LIN {X 0,Y 525.435,Z 278.246,A -85,B 0,C 180,E1 -4754.99,E2 -4754.99} C_VEL
LIN {X 0,Y 525.931,Z 282.457,A -85,B 0,C 180,E1 -4755.064,E2 -4755.064} C_VEL
LIN {X 0,Y 525.504,Z 378.759,A -85,B 0,C 180,E1 -4756.414,E2 -4756.414} C_VEL
LIN {X 0,Y 525.272,Z 391.955,A -85,B 0,C 180,E1 -4756.753,E2 -4756.753} C_VEL
LIN {X 0,Y 525.033,Z 404.647,A -85,B 0,C 180,E1 -4757.239,E2 -4757.239} C_VEL
LIN {X 0,Y 524.762,Z 415.969,A -85,B 0,C 180,E1 -4757.824,E2 -4757.824} C_VEL
LIN {X 0,Y 524.543,Z 427.589,A -85,B 0,C 180,E1 -4758.601,E2 -4758.601} C_VEL
LIN {X 0,Y 524.212,Z 438.073,A -85,B 0,C 180,E1 -4759.474,E2 -4759.474} C_VEL
LIN {X 0,Y 524.018,Z 446.642,A -85,B 0,C 180,E1 -4760.348,E2 -4760.348} C_VEL
LIN {X 0,Y 523.819,Z 454.543,A -85,B 0,C 180,E1 -4761.317,E2 -4761.317} C_VEL
LIN {X 0,Y 523.627,Z 462.256,A -85,B 0,C 180,E1 -4762.479,E2 -4762.479} C_VEL
LIN {X 0,Y 523.496,Z 469.355,A -85,B 0,C 180,E1 -4763.833,E2 -4763.833} C_VEL
LIN {X 0,Y 523.385,Z 474.077,A -85,B 0,C 180,E1 -4764.992,E2 -4764.992} C_VEL
LIN {X 0,Y 523.446,Z 477.686,A -85,B 0,C 180,E1 -4766.149,E2 -4766.149} C_VEL
LIN {X 0,Y 523.37,Z 479.546,A -85,B 0,C 180,E1 -4766.92,E2 -4766.92} C_VEL
LIN {X 0,Y 523.336,Z 480.94,A -85,B 0,C 180,E1 -4767.69,E2 -4767.69} C_VEL
LIN {X 0,Y 523.251,Z 482.541,A -85,B 0,C 180,E1 -4769.229,E2 -4769.229} C_VEL
LIN {X 0,Y 523.248,Z 482.758,A -85,B 0,C 180,E1 -4769.999,E2 -4769.999} C_VEL
LIN {X 0,Y 523.275,Z 481.936,A -85,B 0,C 180,E1 -4771.538,E2 -4771.538} C_VEL
LIN {X 0,Y 523.336,Z 480.943,A -85,B 0,C 180,E1 -4772.308,E2 -4772.308} C_VEL
LIN {X 0,Y 523.369,Z 479.548,A -85,B 0,C 180,E1 -4773.078,E2 -4773.078} C_VEL
LIN {X 0,Y 523.425,Z 476.616,A -85,B 0,C 180,E1 -4774.234,E2 -4774.234} C_VEL
LIN {X 0,Y 523.461,Z 472.643,A -85,B 0,C 180,E1 -4775.391,E2 -4775.391} C_VEL
LIN {X 0,Y 523.504,Z 466.574,A -85,B 0,C 180,E1 -4776.736,E2 -4776.736} C_VEL
LIN {X 0,Y 523.675,Z 459.848,A -85,B 0,C 180,E1 -4777.905,E2 -4777.905} C_VEL
LIN {X 0,Y 523.855,Z 451.549,A -85,B 0,C 180,E1 -4779.068,E2 -4779.068} C_VEL
LIN {X 0,Y 524.068,Z 443.032,A -85,B 0,C 180,E1 -4780.039,E2 -4780.039} C_VEL
LIN {X 0,Y 524.349,Z 432.504,A -85,B 0,C 180,E1 -4781.009,E2 -4781.009} C_VEL
LIN {X 0,Y 524.658,Z 422.256,A -85,B 0,C 180,E1 -4781.774,E2 -4781.774} C_VEL
LIN {X 0,Y 524.908,Z 410.629,A -85,B 0,C 180,E1 -4782.467,E2 -4782.467} C_VEL
LIN {X 0,Y 525.182,Z 398.8,A -85,B 0,C 180,E1 -4783,E2 -4783} C_VEL
LIN {X 0,Y 525.389,Z 386.064,A -85,B 0,C 180,E1 -4783.413,E2 -4783.413} C_VEL
LIN {X 0,Y 525.543,Z 372.951,A -85,B 0,C 180,E1 -4783.68,E2 -4783.68} C_VEL
LIN {X 0,Y 525.872,Z 280.781,A -85,B 0,C 180,E1 -4784.959,E2 -4784.959} C_VEL
LIN {X 0,Y 524.29,Z 270.778,A -85,B 0,C 180,E1 -4785.168,E2 -4785.168} C_VEL
LIN {X 0,Y 524.631,Z 252.415,A -85,B 0,C 180,E1 -4788.125,E2 -4788.125} C_VEL
LIN {X 0,Y 525.085,Z 232.615,A -85,B 0,C 180,E1 -4791.389,E2 -4791.389} C_VEL
LIN {X 0,Y 524.921,Z 226.943,A -85,B 0,C 180,E1 -4792.346,E2 -4792.346} C_VEL
LIN {X 0,Y 524.015,Z 222.139,A -85,B 0,C 180,E1 -4793.2,E2 -4793.2} C_VEL
LIN {X 0,Y 523.924,Z 221.726,A -85,B 0,C 180,E1 -4793.414,E2 -4793.414} C_VEL
LIN {X 0,Y 523.946,Z 221.719,A -85,B 0,C 180,E1 -4796.271,E2 -4796.271} C_VEL
LIN {X 0,Y 523.933,Z 221.718,A -85,B 0,C 180,E1 -4798.873,E2 -4798.873} C_VEL
LIN {X 0,Y 523.923,Z 221.722,A -85,B 0,C 180,E1 -4801.542,E2 -4801.542} C_VEL
LIN {X 0,Y 523.934,Z 221.721,A -85,B 0,C 180,E1 -4804.288,E2 -4804.288} C_VEL
LIN {X 0,Y 523.906,Z 221.721,A -85,B 0,C 180,E1 -4807.13,E2 -4807.13} C_VEL
LIN {X 0,Y 523.915,Z 221.727,A -85,B 0,C 180,E1 -4810.124,E2 -4810.124} C_VEL
LIN {X 0,Y 523.887,Z 221.721,A -85,B 0,C 180,E1 -4813.168,E2 -4813.168} C_VEL
LIN {X 0,Y 523.919,Z 221.721,A -85,B 0,C 180,E1 -4815.767,E2 -4815.767} C_VEL
LIN {X 0,Y 523.896,Z 221.723,A -85,B 0,C 180,E1 -4818.9,E2 -4818.9} C_VEL
LIN {X 0,Y 523.899,Z 221.723,A -85,B 0,C 180,E1 -4821.894,E2 -4821.894} C_VEL
LIN {X 0,Y 523.914,Z 221.722,A -85,B 0,C 180,E1 -4824.909,E2 -4824.909} C_VEL
LIN {X 0,Y 523.929,Z 221.716,A -85,B 0,C 180,E1 -4827.677,E2 -4827.677} C_VEL
LIN {X 0,Y 523.932,Z 221.724,A -85,B 0,C 180,E1 -4830.677,E2 -4830.677} C_VEL
LIN {X 0,Y 523.893,Z 221.719,A -85,B 0,C 180,E1 -4833.721,E2 -4833.721} C_VEL
LIN {X 0,Y 523.889,Z 221.725,A -85,B 0,C 180,E1 -4836.265,E2 -4836.265} C_VEL
LIN {X 0,Y 523.908,Z 221.729,A -85,B 0,C 180,E1 -4838.761,E2 -4838.761} C_VEL
LIN {X 0,Y 523.907,Z 221.723,A -85,B 0,C 180,E1 -4841.215,E2 -4841.215} C_VEL
LIN {X 0,Y 523.867,Z 221.724,A -85,B 0,C 180,E1 -4843.633,E2 -4843.633} C_VEL
LIN {X 0,Y 523.95,Z 221.719,A -85,B 0,C 180,E1 -4845.231,E2 -4845.231} C_VEL
LIN {X 0,Y 523.983,Z 221.71,A -85,B 0,C 180,E1 -4848.389,E2 -4848.389} C_VEL
LIN {X 0,Y 523.936,Z 221.719,A -85,B 0,C 180,E1 -4851.51,E2 -4851.51} C_VEL
LIN {X 0,Y 523.997,Z 221.708,A -85,B 0,C 180,E1 -4853.836,E2 -4853.836} C_VEL
LIN {X 0,Y 524.014,Z 221.712,A -85,B 0,C 180,E1 -4856.92,E2 -4856.92} C_VEL
LIN {X 0,Y 524.088,Z 221.697,A -85,B 0,C 180,E1 -4859.995,E2 -4859.995} C_VEL
LIN {X 0,Y 524.048,Z 221.707,A -85,B 0,C 180,E1 -4863.07,E2 -4863.07} C_VEL
LIN {X 0,Y 524.011,Z 221.708,A -85,B 0,C 180,E1 -4866.154,E2 -4866.154} C_VEL
LIN {X 0,Y 523.979,Z 221.711,A -85,B 0,C 180,E1 -4868.479,E2 -4868.479} C_VEL
LIN {X 0,Y 523.997,Z 221.716,A -85,B 0,C 180,E1 -4871.746,E2 -4871.746} C_VEL
LIN {X 0,Y 523.963,Z 221.715,A -85,B 0,C 180,E1 -4875.048,E2 -4875.048} C_VEL
LIN {X 0,Y 523.931,Z 221.724,A -85,B 0,C 180,E1 -4877.964,E2 -4877.964} C_VEL
LIN {X 0,Y 523.938,Z 221.718,A -85,B 0,C 180,E1 -4880.405,E2 -4880.405} C_VEL
LIN {X 0,Y 523.927,Z 221.72,A -85,B 0,C 180,E1 -4882.886,E2 -4882.886} C_VEL
LIN {X 0,Y 524.021,Z 221.823,A -85,B 0,C 180,E1 -4884.93,E2 -4884.93} C_VEL
LIN {X 0,Y 524.568,Z 226.394,A -85,B 0,C 180,E1 -4885.76,E2 -4885.76} C_VEL
LIN {X 0,Y 524.321,Z 244.865,A -85,B 0,C 180,E1 -4888.844,E2 -4888.844} C_VEL
LIN {X 0,Y 524.2,Z 257.025,A -85,B 0,C 180,E1 -4890.872,E2 -4890.872} C_VEL
LIN {X 0,Y 525.251,Z 263.257,A -85,B 0,C 180,E1 -4891.016,E2 -4891.016} C_VEL
LIN {X 0,Y 525.911,Z 268.568,A -85,B 0,C 180,E1 -4891.111,E2 -4891.111} C_VEL
LIN {X 0,Y 525.501,Z 364.681,A -85,B 0,C 180,E1 -4892.465,E2 -4892.465} C_VEL
LIN {X 0,Y 525.441,Z 368.257,A -85,B 0,C 180,E1 -4892.54,E2 -4892.54} C_VEL
LIN {X 0,Y 524.652,Z 374.018,A -85,B 0,C 180,E1 -4892.662,E2 -4892.662} C_VEL
LIN {X 0,Y 521.72,Z 383.263,A -85,B 0,C 180,E1 -4892.894,E2 -4892.894} C_VEL
LIN {X 0,Y 518.781,Z 392.251,A -85,B 0,C 180,E1 -4893.214,E2 -4893.214} C_VEL
LIN {X 0,Y 517.98,Z 397.6,A -85,B 0,C 180,E1 -4893.474,E2 -4893.474} C_VEL
LIN {X 0,Y 517.687,Z 409.287,A -85,B 0,C 180,E1 -4894.194,E2 -4894.194} C_VEL
LIN {X 0,Y 517.367,Z 419.582,A -85,B 0,C 180,E1 -4894.992,E2 -4894.992} C_VEL
LIN {X 0,Y 517.046,Z 430.003,A -85,B 0,C 180,E1 -4895.997,E2 -4895.997} C_VEL
LIN {X 0,Y 516.831,Z 438.296,A -85,B 0,C 180,E1 -4896.984,E2 -4896.984} C_VEL
LIN {X 0,Y 516.612,Z 445.81,A -85,B 0,C 180,E1 -4898.073,E2 -4898.073} C_VEL
LIN {X 0,Y 516.482,Z 451.883,A -85,B 0,C 180,E1 -4899.141,E2 -4899.141} C_VEL
LIN {X 0,Y 516.356,Z 457.376,A -85,B 0,C 180,E1 -4900.344,E2 -4900.344} C_VEL
LIN {X 0,Y 516.321,Z 461.562,A -85,B 0,C 180,E1 -4901.53,E2 -4901.53} C_VEL
LIN {X 0,Y 516.21,Z 465.087,A -85,B 0,C 180,E1 -4902.89,E2 -4902.89} C_VEL
LIN {X 0,Y 516.174,Z 466.943,A -85,B 0,C 180,E1 -4903.968,E2 -4903.968} C_VEL
LIN {X 0,Y 516.209,Z 468.031,A -85,B 0,C 180,E1 -4905.058,E2 -4905.058} C_VEL
LIN {X 0,Y 516.152,Z 468.339,A -85,B 0,C 180,E1 -4906.18,E2 -4906.18} C_VEL
LIN {X 0,Y 516.171,Z 467.809,A -85,B 0,C 180,E1 -4907.316,E2 -4907.316} C_VEL
LIN {X 0,Y 516.222,Z 466.397,A -85,B 0,C 180,E1 -4908.473,E2 -4908.473} C_VEL
LIN {X 0,Y 516.237,Z 464.011,A -85,B 0,C 180,E1 -4909.662,E2 -4909.662} C_VEL
LIN {X 0,Y 516.31,Z 460.568,A -85,B 0,C 180,E1 -4910.872,E2 -4910.872} C_VEL
LIN {X 0,Y 516.422,Z 455.246,A -85,B 0,C 180,E1 -4912.239,E2 -4912.239} C_VEL
LIN {X 0,Y 516.534,Z 449.57,A -85,B 0,C 180,E1 -4913.38,E2 -4913.38} C_VEL
LIN {X 0,Y 516.757,Z 441.466,A -85,B 0,C 180,E1 -4914.673,E2 -4914.673} C_VEL
LIN {X 0,Y 516.984,Z 432.284,A -85,B 0,C 180,E1 -4915.838,E2 -4915.838} C_VEL
LIN {X 0,Y 517.282,Z 422.326,A -85,B 0,C 180,E1 -4916.851,E2 -4916.851} C_VEL
LIN {X 0,Y 517.578,Z 412.074,A -85,B 0,C 180,E1 -4917.694,E2 -4917.694} C_VEL
LIN {X 0,Y 517.887,Z 401.265,A -85,B 0,C 180,E1 -4918.412,E2 -4918.412} C_VEL
LIN {X 0,Y 518.157,Z 390.366,A -85,B 0,C 180,E1 -4918.977,E2 -4918.977} C_VEL
LIN {X 0,Y 518.381,Z 377.647,A -85,B 0,C 180,E1 -4919.472,E2 -4919.472} C_VEL
LIN {X 0,Y 518.585,Z 364.695,A -85,B 0,C 180,E1 -4919.809,E2 -4919.809} C_VEL
LIN {X 0,Y 518.901,Z 266.997,A -85,B 0,C 180,E1 -4921.208,E2 -4921.208} C_VEL
LIN {X 0,Y 517.258,Z 257.639,A -85,B 0,C 180,E1 -4921.413,E2 -4921.413} C_VEL
LIN {X 0,Y 517.338,Z 254.175,A -85,B 0,C 180,E1 -4921.99,E2 -4921.99} C_VEL
LIN {X 0,Y 517.766,Z 237.292,A -85,B 0,C 180,E1 -4925.118,E2 -4925.118} C_VEL
LIN {X 0,Y 517.886,Z 228.224,A -85,B 0,C 180,E1 -4926.826,E2 -4926.826} C_VEL
LIN {X 0,Y 516.929,Z 222.738,A -85,B 0,C 180,E1 -4927.942,E2 -4927.942} C_VEL
LIN {X 0,Y 516.829,Z 222.606,A -85,B 0,C 180,E1 -4930.954,E2 -4930.954} C_VEL
LIN {X 0,Y 516.846,Z 222.599,A -85,B 0,C 180,E1 -4933.41,E2 -4933.41} C_VEL
LIN {X 0,Y 516.848,Z 222.599,A -85,B 0,C 180,E1 -4935.834,E2 -4935.834} C_VEL
LIN {X 0,Y 516.924,Z 222.593,A -85,B 0,C 180,E1 -4938.234,E2 -4938.234} C_VEL
LIN {X 0,Y 516.899,Z 222.593,A -85,B 0,C 180,E1 -4941.4,E2 -4941.4} C_VEL
LIN {X 0,Y 516.992,Z 222.585,A -85,B 0,C 180,E1 -4944.541,E2 -4944.541} C_VEL
LIN {X 0,Y 517.007,Z 222.579,A -85,B 0,C 180,E1 -4947.664,E2 -4947.664} C_VEL
LIN {X 0,Y 517.022,Z 222.582,A -85,B 0,C 180,E1 -4950.78,E2 -4950.78} C_VEL
LIN {X 0,Y 516.976,Z 222.592,A -85,B 0,C 180,E1 -4953.118,E2 -4953.118} C_VEL
LIN {X 0,Y 516.94,Z 222.587,A -85,B 0,C 180,E1 -4956.245,E2 -4956.245} C_VEL
LIN {X 0,Y 516.893,Z 222.602,A -85,B 0,C 180,E1 -4959.392,E2 -4959.392} C_VEL
LIN {X 0,Y 516.908,Z 222.594,A -85,B 0,C 180,E1 -4961.827,E2 -4961.827} C_VEL
LIN {X 0,Y 516.885,Z 222.598,A -85,B 0,C 180,E1 -4965.156,E2 -4965.156} C_VEL
LIN {X 0,Y 516.854,Z 222.599,A -85,B 0,C 180,E1 -4968.226,E2 -4968.226} C_VEL
LIN {X 0,Y 516.843,Z 222.599,A -85,B 0,C 180,E1 -4970.705,E2 -4970.705} C_VEL
LIN {X 0,Y 516.811,Z 222.605,A -85,B 0,C 180,E1 -4973.227,E2 -4973.227} C_VEL
LIN {X 0,Y 516.884,Z 222.599,A -85,B 0,C 180,E1 -4976.202,E2 -4976.202} C_VEL
LIN {X 0,Y 516.874,Z 222.596,A -85,B 0,C 180,E1 -4979.309,E2 -4979.309} C_VEL
LIN {X 0,Y 516.843,Z 222.602,A -85,B 0,C 180,E1 -4982.55,E2 -4982.55} C_VEL
LIN {X 0,Y 516.827,Z 222.601,A -85,B 0,C 180,E1 -4985.338,E2 -4985.338} C_VEL
LIN {X 0,Y 516.828,Z 222.605,A -85,B 0,C 180,E1 -4987.949,E2 -4987.949} C_VEL
LIN {X 0,Y 516.858,Z 222.601,A -85,B 0,C 180,E1 -4990.745,E2 -4990.745} C_VEL
LIN {X 0,Y 516.836,Z 222.601,A -85,B 0,C 180,E1 -4993.909,E2 -4993.909} C_VEL
LIN {X 0,Y 516.839,Z 222.602,A -85,B 0,C 180,E1 -4996.113,E2 -4996.113} C_VEL
LIN {X 0,Y 516.869,Z 222.597,A -85,B 0,C 180,E1 -4999.267,E2 -4999.267} C_VEL
LIN {X 0,Y 516.845,Z 222.599,A -85,B 0,C 180,E1 -5002.063,E2 -5002.063} C_VEL
LIN {X 0,Y 516.857,Z 222.602,A -85,B 0,C 180,E1 -5005.182,E2 -5005.182} C_VEL
LIN {X 0,Y 516.844,Z 222.598,A -85,B 0,C 180,E1 -5007.982,E2 -5007.982} C_VEL
LIN {X 0,Y 516.895,Z 222.596,A -85,B 0,C 180,E1 -5010.702,E2 -5010.702} C_VEL
LIN {X 0,Y 516.919,Z 222.591,A -85,B 0,C 180,E1 -5013.811,E2 -5013.811} C_VEL
LIN {X 0,Y 516.847,Z 222.601,A -85,B 0,C 180,E1 -5016.783,E2 -5016.783} C_VEL
LIN {X 0,Y 516.924,Z 222.593,A -85,B 0,C 180,E1 -5019.738,E2 -5019.738} C_VEL
LIN {X 0,Y 516.893,Z 222.592,A -85,B 0,C 180,E1 -5022.602,E2 -5022.602} C_VEL
LIN {X 0,Y 516.933,Z 222.59,A -85,B 0,C 180,E1 -5025.036,E2 -5025.036} C_VEL
LIN {X 0,Y 516.961,Z 222.586,A -85,B 0,C 180,E1 -5028.24,E2 -5028.24} C_VEL
LIN {X 0,Y 516.96,Z 222.588,A -85,B 0,C 180,E1 -5031.405,E2 -5031.405} C_VEL
LIN {X 0,Y 516.994,Z 222.581,A -85,B 0,C 180,E1 -5034.545,E2 -5034.545} C_VEL
LIN {X 0,Y 517.081,Z 222.574,A -85,B 0,C 180,E1 -5037.668,E2 -5037.668} C_VEL
LIN {X 0,Y 517.072,Z 222.571,A -85,B 0,C 180,E1 -5040.784,E2 -5040.784} C_VEL
LIN {X 0,Y 516.952,Z 222.585,A -85,B 0,C 180,E1 -5043.122,E2 -5043.122} C_VEL
LIN {X 0,Y 516.979,Z 222.592,A -85,B 0,C 180,E1 -5046.248,E2 -5046.248} C_VEL
LIN {X 0,Y 516.926,Z 222.588,A -85,B 0,C 180,E1 -5049.394,E2 -5049.394} C_VEL
LIN {X 0,Y 516.965,Z 222.585,A -85,B 0,C 180,E1 -5051.811,E2 -5051.811} C_VEL
LIN {X 0,Y 516.951,Z 222.587,A -85,B 0,C 180,E1 -5055.146,E2 -5055.146} C_VEL
LIN {X 0,Y 516.926,Z 222.591,A -85,B 0,C 180,E1 -5058.226,E2 -5058.226} C_VEL
LIN {X 0,Y 516.917,Z 222.599,A -85,B 0,C 180,E1 -5060.705,E2 -5060.705} C_VEL
LIN {X 0,Y 516.872,Z 222.599,A -85,B 0,C 180,E1 -5063.227,E2 -5063.227} C_VEL
LIN {X 0,Y 516.898,Z 222.592,A -85,B 0,C 180,E1 -5066.184,E2 -5066.184} C_VEL
LIN {X 0,Y 516.921,Z 222.595,A -85,B 0,C 180,E1 -5069.308,E2 -5069.308} C_VEL
LIN {X 0,Y 516.91,Z 222.592,A -85,B 0,C 180,E1 -5072.544,E2 -5072.544} C_VEL
LIN {X 0,Y 516.872,Z 222.604,A -85,B 0,C 180,E1 -5075.329,E2 -5075.329} C_VEL
LIN {X 0,Y 516.895,Z 222.594,A -85,B 0,C 180,E1 -5077.944,E2 -5077.944} C_VEL
LIN {X 0,Y 516.868,Z 222.596,A -85,B 0,C 180,E1 -5080.746,E2 -5080.746} C_VEL
LIN {X 0,Y 516.878,Z 222.599,A -85,B 0,C 180,E1 -5083.907,E2 -5083.907} C_VEL
LIN {X 0,Y 516.878,Z 222.597,A -85,B 0,C 180,E1 -5086.111,E2 -5086.111} C_VEL
LIN {X 0,Y 516.868,Z 222.598,A -85,B 0,C 180,E1 -5089.256,E2 -5089.256} C_VEL
LIN {X 0,Y 516.881,Z 222.6,A -85,B 0,C 180,E1 -5092.06,E2 -5092.06} C_VEL
LIN {X 0,Y 516.889,Z 222.593,A -85,B 0,C 180,E1 -5095.175,E2 -5095.175} C_VEL
LIN {X 0,Y 516.888,Z 222.602,A -85,B 0,C 180,E1 -5097.975,E2 -5097.975} C_VEL
LIN {X 0,Y 516.935,Z 222.591,A -85,B 0,C 180,E1 -5100.695,E2 -5100.695} C_VEL
LIN {X 0,Y 516.91,Z 222.598,A -85,B 0,C 180,E1 -5103.815,E2 -5103.815} C_VEL
LIN {X 0,Y 516.917,Z 222.681,A -85,B 0,C 180,E1 -5106.353,E2 -5106.353} C_VEL
LIN {X 0,Y 518.165,Z 229.675,A -85,B 0,C 180,E1 -5107.679,E2 -5107.679} C_VEL
LIN {X 0,Y 518.072,Z 239.332,A -85,B 0,C 180,E1 -5109.346,E2 -5109.346} C_VEL
LIN {X 0,Y 517.604,Z 257.547,A -85,B 0,C 180,E1 -5112.433,E2 -5112.433} C_VEL
LIN {X 0,Y 517.3,Z 270.913,A -85,B 0,C 180,E1 -5114.625,E2 -5114.625} C_VEL
LIN {X 0,Y 519.083,Z 282.681,A -85,B 0,C 180,E1 -5114.868,E2 -5114.868} C_VEL
LIN {X 0,Y 518.605,Z 378.458,A -85,B 0,C 180,E1 -5116.23,E2 -5116.23} C_VEL
LIN {X 0,Y 518.357,Z 391.716,A -85,B 0,C 180,E1 -5116.573,E2 -5116.573} C_VEL
LIN {X 0,Y 518.08,Z 404.443,A -85,B 0,C 180,E1 -5117.065,E2 -5117.065} C_VEL
LIN {X 0,Y 517.821,Z 415.805,A -85,B 0,C 180,E1 -5117.659,E2 -5117.659} C_VEL
LIN {X 0,Y 517.564,Z 427.432,A -85,B 0,C 180,E1 -5118.445,E2 -5118.445} C_VEL
LIN {X 0,Y 517.202,Z 437.928,A -85,B 0,C 180,E1 -5119.329,E2 -5119.329} C_VEL
LIN {X 0,Y 516.97,Z 446.506,A -85,B 0,C 180,E1 -5120.215,E2 -5120.215} C_VEL
LIN {X 0,Y 516.741,Z 454.415,A -85,B 0,C 180,E1 -5121.198,E2 -5121.198} C_VEL
LIN {X 0,Y 516.555,Z 462.138,A -85,B 0,C 180,E1 -5122.376,E2 -5122.376} C_VEL
LIN {X 0,Y 516.408,Z 469.243,A -85,B 0,C 180,E1 -5123.748,E2 -5123.748} C_VEL
LIN {X 0,Y 516.315,Z 473.971,A -85,B 0,C 180,E1 -5124.923,E2 -5124.923} C_VEL
LIN {X 0,Y 516.354,Z 477.583,A -85,B 0,C 180,E1 -5126.096,E2 -5126.096} C_VEL
LIN {X 0,Y 516.285,Z 479.445,A -85,B 0,C 180,E1 -5126.877,E2 -5126.877} C_VEL
LIN {X 0,Y 516.263,Z 480.841,A -85,B 0,C 180,E1 -5127.658,E2 -5127.658} C_VEL
LIN {X 0,Y 516.161,Z 482.443,A -85,B 0,C 180,E1 -5129.219,E2 -5129.219} C_VEL
LIN {X 0,Y 516.156,Z 482.66,A -85,B 0,C 180,E1 -5129.999,E2 -5129.999} C_VEL
LIN {X 0,Y 516.193,Z 481.837,A -85,B 0,C 180,E1 -5131.559,E2 -5131.559} C_VEL
LIN {X 0,Y 516.262,Z 480.842,A -85,B 0,C 180,E1 -5132.339,E2 -5132.339} C_VEL
LIN {X 0,Y 516.284,Z 479.445,A -85,B 0,C 180,E1 -5133.12,E2 -5133.12} C_VEL
LIN {X 0,Y 516.314,Z 476.508,A -85,B 0,C 180,E1 -5134.292,E2 -5134.292} C_VEL
LIN {X 0,Y 516.398,Z 472.531,A -85,B 0,C 180,E1 -5135.465,E2 -5135.465} C_VEL
LIN {X 0,Y 516.421,Z 467.33,A -85,B 0,C 180,E1 -5136.658,E2 -5136.658} C_VEL
LIN {X 0,Y 516.584,Z 460.955,A -85,B 0,C 180,E1 -5137.818,E2 -5137.818} C_VEL
LIN {X 0,Y 516.769,Z 452.905,A -85,B 0,C 180,E1 -5138.996,E2 -5138.996} C_VEL
LIN {X 0,Y 517.013,Z 444.694,A -85,B 0,C 180,E1 -5139.979,E2 -5139.979} C_VEL
LIN {X 0,Y 517.319,Z 434.672,A -85,B 0,C 180,E1 -5140.963,E2 -5140.963} C_VEL
LIN {X 0,Y 517.646,Z 424.759,A -85,B 0,C 180,E1 -5141.749,E2 -5141.749} C_VEL
LIN {X 0,Y 517.856,Z 413.549,A -85,B 0,C 180,E1 -5142.464,E2 -5142.464} C_VEL
LIN {X 0,Y 518.161,Z 400.984,A -85,B 0,C 180,E1 -5143.08,E2 -5143.08} C_VEL
LIN {X 0,Y 518.441,Z 388.51,A -85,B 0,C 180,E1 -5143.522,E2 -5143.522} C_VEL
LIN {X 0,Y 518.602,Z 375.529,A -85,B 0,C 180,E1 -5143.817,E2 -5143.817} C_VEL
LIN {X 0,Y 518.925,Z 280.883,A -85,B 0,C 180,E1 -5145.161,E2 -5145.161} C_VEL
LIN {X 0,Y 517.252,Z 270.718,A -85,B 0,C 180,E1 -5145.375,E2 -5145.375} C_VEL
LIN {X 0,Y 517.636,Z 253.385,A -85,B 0,C 180,E1 -5148.195,E2 -5148.195} C_VEL
LIN {X 0,Y 518.119,Z 233.686,A -85,B 0,C 180,E1 -5151.482,E2 -5151.482} C_VEL
LIN {X 0,Y 518.014,Z 228.739,A -85,B 0,C 180,E1 -5152.325,E2 -5152.325} C_VEL
LIN {X 0,Y 516.905,Z 222.749,A -85,B 0,C 180,E1 -5153.432,E2 -5153.432} C_VEL
LIN {X 0,Y 516.914,Z 222.594,A -85,B 0,C 180,E1 -5156.656,E2 -5156.656} C_VEL
LIN {X 0,Y 516.912,Z 222.597,A -85,B 0,C 180,E1 -5159.521,E2 -5159.521} C_VEL
LIN {X 0,Y 516.899,Z 222.595,A -85,B 0,C 180,E1 -5162.541,E2 -5162.541} C_VEL
LIN {X 0,Y 516.866,Z 222.599,A -85,B 0,C 180,E1 -5165.326,E2 -5165.326} C_VEL
LIN {X 0,Y 516.88,Z 222.603,A -85,B 0,C 180,E1 -5167.94,E2 -5167.94} C_VEL
LIN {X 0,Y 516.856,Z 222.599,A -85,B 0,C 180,E1 -5170.742,E2 -5170.742} C_VEL
LIN {X 0,Y 516.882,Z 222.6,A -85,B 0,C 180,E1 -5173.901,E2 -5173.901} C_VEL
LIN {X 0,Y 516.881,Z 222.602,A -85,B 0,C 180,E1 -5176.104,E2 -5176.104} C_VEL
LIN {X 0,Y 516.852,Z 222.599,A -85,B 0,C 180,E1 -5179.252,E2 -5179.252} C_VEL
LIN {X 0,Y 516.859,Z 222.602,A -85,B 0,C 180,E1 -5182.057,E2 -5182.057} C_VEL
LIN {X 0,Y 516.87,Z 222.597,A -85,B 0,C 180,E1 -5185.171,E2 -5185.171} C_VEL
LIN {X 0,Y 516.865,Z 222.598,A -85,B 0,C 180,E1 -5187.971,E2 -5187.971} C_VEL
LIN {X 0,Y 516.899,Z 222.6,A -85,B 0,C 180,E1 -5190.69,E2 -5190.69} C_VEL
LIN {X 0,Y 516.874,Z 222.593,A -85,B 0,C 180,E1 -5193.815,E2 -5193.815} C_VEL
LIN {X 0,Y 516.834,Z 222.607,A -85,B 0,C 180,E1 -5196.771,E2 -5196.771} C_VEL
LIN {X 0,Y 516.871,Z 222.596,A -85,B 0,C 180,E1 -5199.746,E2 -5199.746} C_VEL
LIN {X 0,Y 516.867,Z 222.602,A -85,B 0,C 180,E1 -5202.59,E2 -5202.59} C_VEL
LIN {X 0,Y 516.92,Z 222.598,A -85,B 0,C 180,E1 -5205.025,E2 -5205.025} C_VEL
LIN {X 0,Y 516.956,Z 222.584,A -85,B 0,C 180,E1 -5208.229,E2 -5208.229} C_VEL
LIN {X 0,Y 516.91,Z 222.595,A -85,B 0,C 180,E1 -5211.394,E2 -5211.394} C_VEL
LIN {X 0,Y 516.967,Z 222.584,A -85,B 0,C 180,E1 -5213.752,E2 -5213.752} C_VEL
LIN {X 0,Y 516.956,Z 222.591,A -85,B 0,C 180,E1 -5216.878,E2 -5216.878} C_VEL
LIN {X 0,Y 517.077,Z 222.579,A -85,B 0,C 180,E1 -5219.216,E2 -5219.216} C_VEL
LIN {X 0,Y 517.057,Z 222.572,A -85,B 0,C 180,E1 -5222.332,E2 -5222.332} C_VEL
LIN {X 0,Y 517.003,Z 222.589,A -85,B 0,C 180,E1 -5225.455,E2 -5225.455} C_VEL
LIN {X 0,Y 516.944,Z 222.588,A -85,B 0,C 180,E1 -5228.595,E2 -5228.595} C_VEL
LIN {X 0,Y 516.956,Z 222.592,A -85,B 0,C 180,E1 -5231.819,E2 -5231.819} C_VEL
LIN {X 0,Y 516.916,Z 222.594,A -85,B 0,C 180,E1 -5235.142,E2 -5235.142} C_VEL
LIN {X 0,Y 516.892,Z 222.598,A -85,B 0,C 180,E1 -5238.217,E2 -5238.217} C_VEL
LIN {X 0,Y 516.881,Z 222.596,A -85,B 0,C 180,E1 -5240.696,E2 -5240.696} C_VEL
LIN {X 0,Y 516.873,Z 222.601,A -85,B 0,C 180,E1 -5243.216,E2 -5243.216} C_VEL
LIN {X 0,Y 516.975,Z 222.758,A -85,B 0,C 180,E1 -5244.83,E2 -5244.83} C_VEL
LIN {X 0,Y 517.609,Z 227.905,A -85,B 0,C 180,E1 -5245.745,E2 -5245.745} C_VEL
LIN {X 0,Y 517.322,Z 247.436,A -85,B 0,C 180,E1 -5249.049,E2 -5249.049} C_VEL
LIN {X 0,Y 517.201,Z 256.999,A -85,B 0,C 180,E1 -5250.655,E2 -5250.655} C_VEL
LIN {X 0,Y 517.806,Z 260.606,A -85,B 0,C 180,E1 -5250.757,E2 -5250.757} C_VEL
LIN {X 0,Y 519.054,Z 267.977,A -85,B 0,C 180,E1 -5250.901,E2 -5250.901} C_VEL
LIN {X 0,Y 518.582,Z 365.471,A -85,B 0,C 180,E1 -5252.299,E2 -5252.299} C_VEL
LIN {X 0,Y 518.376,Z 378.677,A -85,B 0,C 180,E1 -5252.653,E2 -5252.653} C_VEL
LIN {X 0,Y 518.169,Z 390.88,A -85,B 0,C 180,E1 -5253.137,E2 -5253.137} C_VEL
LIN {X 0,Y 517.98,Z 397.6,A -85,B 0,C 180,E1 -5253.474,E2 -5253.474} C_VEL
LIN {X 0,Y 517.164,Z 402.918,A -85,B 0,C 180,E1 -5253.761,E2 -5253.761} C_VEL
LIN {X 0,Y 514.133,Z 411.278,A -85,B 0,C 180,E1 -5254.252,E2 -5254.252} C_VEL
LIN {X 0,Y 511.101,Z 419.182,A -85,B 0,C 180,E1 -5254.817,E2 -5254.817} C_VEL
LIN {X 0,Y 510.279,Z 423.76,A -85,B 0,C 180,E1 -5255.218,E2 -5255.218} C_VEL
LIN {X 0,Y 509.976,Z 432.598,A -85,B 0,C 180,E1 -5256.143,E2 -5256.143} C_VEL
LIN {X 0,Y 509.69,Z 441.865,A -85,B 0,C 180,E1 -5257.342,E2 -5257.342} C_VEL
LIN {X 0,Y 509.495,Z 449.696,A -85,B 0,C 180,E1 -5258.612,E2 -5258.612} C_VEL
LIN {X 0,Y 509.319,Z 455.979,A -85,B 0,C 180,E1 -5259.904,E2 -5259.904} C_VEL
LIN {X 0,Y 509.251,Z 460.248,A -85,B 0,C 180,E1 -5261.02,E2 -5261.02} C_VEL
LIN {X 0,Y 509.209,Z 462.693,A -85,B 0,C 180,E1 -5261.818,E2 -5261.818} C_VEL
LIN {X 0,Y 509.112,Z 465.46,A -85,B 0,C 180,E1 -5262.979,E2 -5262.979} C_VEL
LIN {X 0,Y 509.086,Z 467.29,A -85,B 0,C 180,E1 -5264.124,E2 -5264.124} C_VEL
LIN {X 0,Y 509.104,Z 468.25,A -85,B 0,C 180,E1 -5265.251,E2 -5265.251} C_VEL
LIN {X 0,Y 509.058,Z 468.402,A -85,B 0,C 180,E1 -5266.349,E2 -5266.349} C_VEL
LIN {X 0,Y 509.073,Z 467.816,A -85,B 0,C 180,E1 -5267.434,E2 -5267.434} C_VEL
LIN {X 0,Y 509.125,Z 466.505,A -85,B 0,C 180,E1 -5268.504,E2 -5268.504} C_VEL
LIN {X 0,Y 509.178,Z 463.207,A -85,B 0,C 180,E1 -5270.075,E2 -5270.075} C_VEL
LIN {X 0,Y 509.223,Z 460.1,A -85,B 0,C 180,E1 -5271.107,E2 -5271.107} C_VEL
LIN {X 0,Y 509.343,Z 455.719,A -85,B 0,C 180,E1 -5272.239,E2 -5272.239} C_VEL
LIN {X 0,Y 509.468,Z 450.204,A -85,B 0,C 180,E1 -5273.379,E2 -5273.379} C_VEL
LIN {X 0,Y 509.68,Z 442.763,A -85,B 0,C 180,E1 -5274.612,E2 -5274.612} C_VEL
LIN {X 0,Y 509.899,Z 434.019,A -85,B 0,C 180,E1 -5275.775,E2 -5275.775} C_VEL
LIN {X 0,Y 510.175,Z 425.319,A -85,B 0,C 180,E1 -5276.721,E2 -5276.721} C_VEL
LIN {X 0,Y 510.541,Z 414.794,A -85,B 0,C 180,E1 -5277.648,E2 -5277.648} C_VEL
LIN {X 0,Y 510.83,Z 404.754,A -85,B 0,C 180,E1 -5278.366,E2 -5278.366} C_VEL
LIN {X 0,Y 511.167,Z 393.137,A -85,B 0,C 180,E1 -5279.023,E2 -5279.023} C_VEL
LIN {X 0,Y 511.412,Z 381.886,A -85,B 0,C 180,E1 -5279.508,E2 -5279.508} C_VEL
LIN {X 0,Y 511.625,Z 369.476,A -85,B 0,C 180,E1 -5279.89,E2 -5279.89} C_VEL
LIN {X 0,Y 511.775,Z 354.011,A -85,B 0,C 180,E1 -5280.166,E2 -5280.166} C_VEL
LIN {X 0,Y 512.082,Z 267.875,A -85,B 0,C 180,E1 -5281.402,E2 -5281.402} C_VEL
LIN {X 0,Y 510.299,Z 257.915,A -85,B 0,C 180,E1 -5281.62,E2 -5281.62} C_VEL
LIN {X 0,Y 510.274,Z 256.485,A -85,B 0,C 180,E1 -5281.802,E2 -5281.802} C_VEL
LIN {X 0,Y 510.809,Z 239.217,A -85,B 0,C 180,E1 -5285.038,E2 -5285.038} C_VEL
LIN {X 0,Y 511.015,Z 230.422,A -85,B 0,C 180,E1 -5286.711,E2 -5286.711} C_VEL
LIN {X 0,Y 509.891,Z 223.803,A -85,B 0,C 180,E1 -5288.048,E2 -5288.048} C_VEL
LIN {X 0,Y 509.833,Z 223.48,A -85,B 0,C 180,E1 -5288.363,E2 -5288.363} C_VEL
LIN {X 0,Y 509.789,Z 223.486,A -85,B 0,C 180,E1 -5290.68,E2 -5290.68} C_VEL
LIN {X 0,Y 509.814,Z 223.476,A -85,B 0,C 180,E1 -5293.174,E2 -5293.174} C_VEL
LIN {X 0,Y 509.813,Z 223.474,A -85,B 0,C 180,E1 -5295.634,E2 -5295.634} C_VEL
LIN {X 0,Y 509.858,Z 223.475,A -85,B 0,C 180,E1 -5298.875,E2 -5298.875} C_VEL
LIN {X 0,Y 509.874,Z 223.468,A -85,B 0,C 180,E1 -5302.079,E2 -5302.079} C_VEL
LIN {X 0,Y 509.938,Z 223.463,A -85,B 0,C 180,E1 -5304.465,E2 -5304.465} C_VEL
LIN {X 0,Y 509.98,Z 223.454,A -85,B 0,C 180,E1 -5307.632,E2 -5307.632} C_VEL
LIN {X 0,Y 509.973,Z 223.454,A -85,B 0,C 180,E1 -5310.001,E2 -5310.001} C_VEL
LIN {X 0,Y 509.917,Z 223.471,A -85,B 0,C 180,E1 -5313.162,E2 -5313.162} C_VEL
LIN {X 0,Y 509.907,Z 223.463,A -85,B 0,C 180,E1 -5316.332,E2 -5316.332} C_VEL
LIN {X 0,Y 509.876,Z 223.468,A -85,B 0,C 180,E1 -5318.722,E2 -5318.722} C_VEL
LIN {X 0,Y 509.877,Z 223.469,A -85,B 0,C 180,E1 -5321.934,E2 -5321.934} C_VEL
LIN {X 0,Y 509.829,Z 223.478,A -85,B 0,C 180,E1 -5325.249,E2 -5325.249} C_VEL
LIN {X 0,Y 509.817,Z 223.478,A -85,B 0,C 180,E1 -5328.005,E2 -5328.005} C_VEL
LIN {X 0,Y 509.781,Z 223.479,A -85,B 0,C 180,E1 -5331.006,E2 -5331.006} C_VEL
LIN {X 0,Y 509.776,Z 223.485,A -85,B 0,C 180,E1 -5333.567,E2 -5333.567} C_VEL
LIN {X 0,Y 509.852,Z 223.472,A -85,B 0,C 180,E1 -5336.385,E2 -5336.385} C_VEL
LIN {X 0,Y 509.823,Z 223.473,A -85,B 0,C 180,E1 -5338.849,E2 -5338.849} C_VEL
LIN {X 0,Y 509.774,Z 223.482,A -85,B 0,C 180,E1 -5341.594,E2 -5341.594} C_VEL
LIN {X 0,Y 509.798,Z 223.482,A -85,B 0,C 180,E1 -5344.419,E2 -5344.419} C_VEL
LIN {X 0,Y 509.765,Z 223.48,A -85,B 0,C 180,E1 -5347.346,E2 -5347.346} C_VEL
LIN {X 0,Y 509.812,Z 223.485,A -85,B 0,C 180,E1 -5350.386,E2 -5350.386} C_VEL
LIN {X 0,Y 509.793,Z 223.479,A -85,B 0,C 180,E1 -5353.07,E2 -5353.07} C_VEL
LIN {X 0,Y 509.786,Z 223.478,A -85,B 0,C 180,E1 -5355.799,E2 -5355.799} C_VEL
LIN {X 0,Y 509.83,Z 223.481,A -85,B 0,C 180,E1 -5358.582,E2 -5358.582} C_VEL
LIN {X 0,Y 509.815,Z 223.474,A -85,B 0,C 180,E1 -5361.669,E2 -5361.669} C_VEL
LIN {X 0,Y 509.811,Z 223.481,A -85,B 0,C 180,E1 -5364.63,E2 -5364.63} C_VEL
LIN {X 0,Y 509.829,Z 223.475,A -85,B 0,C 180,E1 -5367.487,E2 -5367.487} C_VEL
LIN {X 0,Y 509.832,Z 223.472,A -85,B 0,C 180,E1 -5370.28,E2 -5370.28} C_VEL
LIN {X 0,Y 509.859,Z 223.475,A -85,B 0,C 180,E1 -5372.951,E2 -5372.951} C_VEL
LIN {X 0,Y 509.842,Z 223.475,A -85,B 0,C 180,E1 -5375.58,E2 -5375.58} C_VEL
LIN {X 0,Y 509.834,Z 223.476,A -85,B 0,C 180,E1 -5379.005,E2 -5379.005} C_VEL
LIN {X 0,Y 509.847,Z 223.479,A -85,B 0,C 180,E1 -5381.523,E2 -5381.523} C_VEL
LIN {X 0,Y 509.902,Z 223.464,A -85,B 0,C 180,E1 -5384.825,E2 -5384.825} C_VEL
LIN {X 0,Y 509.895,Z 223.467,A -85,B 0,C 180,E1 -5388.13,E2 -5388.13} C_VEL
LIN {X 0,Y 509.906,Z 223.466,A -85,B 0,C 180,E1 -5391.285,E2 -5391.285} C_VEL
LIN {X 0,Y 509.936,Z 223.466,A -85,B 0,C 180,E1 -5393.676,E2 -5393.676} C_VEL
LIN {X 0,Y 509.923,Z 223.461,A -85,B 0,C 180,E1 -5396.845,E2 -5396.845} C_VEL
LIN {X 0,Y 509.932,Z 223.463,A -85,B 0,C 180,E1 -5398.426,E2 -5398.426} C_VEL
LIN {X 0,Y 510.023,Z 223.449,A -85,B 0,C 180,E1 -5400.795,E2 -5400.795} C_VEL
LIN {X 0,Y 510.047,Z 223.451,A -85,B 0,C 180,E1 -5402.374,E2 -5402.374} C_VEL
LIN {X 0,Y 509.956,Z 223.457,A -85,B 0,C 180,E1 -5405.541,E2 -5405.541} C_VEL
LIN {X 0,Y 509.888,Z 223.469,A -85,B 0,C 180,E1 -5408.725,E2 -5408.725} C_VEL
LIN {X 0,Y 509.918,Z 223.464,A -85,B 0,C 180,E1 -5411.936,E2 -5411.936} C_VEL
LIN {X 0,Y 509.91,Z 223.463,A -85,B 0,C 180,E1 -5415.246,E2 -5415.246} C_VEL
LIN {X 0,Y 509.869,Z 223.474,A -85,B 0,C 180,E1 -5418.488,E2 -5418.488} C_VEL
LIN {X 0,Y 509.86,Z 223.475,A -85,B 0,C 180,E1 -5421.005,E2 -5421.005} C_VEL
LIN {X 0,Y 509.834,Z 223.473,A -85,B 0,C 180,E1 -5423.567,E2 -5423.567} C_VEL
LIN {X 0,Y 509.834,Z 223.473,A -85,B 0,C 180,E1 -5426.359,E2 -5426.359} C_VEL
LIN {X 0,Y 509.854,Z 223.476,A -85,B 0,C 180,E1 -5428.849,E2 -5428.849} C_VEL
LIN {X 0,Y 509.83,Z 223.475,A -85,B 0,C 180,E1 -5431.593,E2 -5431.593} C_VEL
LIN {X 0,Y 509.851,Z 223.47,A -85,B 0,C 180,E1 -5434.417,E2 -5434.417} C_VEL
LIN {X 0,Y 509.824,Z 223.483,A -85,B 0,C 180,E1 -5437.344,E2 -5437.344} C_VEL
LIN {X 0,Y 509.831,Z 223.472,A -85,B 0,C 180,E1 -5440.386,E2 -5440.386} C_VEL
LIN {X 0,Y 509.81,Z 223.484,A -85,B 0,C 180,E1 -5443.576,E2 -5443.576} C_VEL
LIN {X 0,Y 509.811,Z 223.475,A -85,B 0,C 180,E1 -5446.426,E2 -5446.426} C_VEL
LIN {X 0,Y 509.831,Z 223.48,A -85,B 0,C 180,E1 -5449.616,E2 -5449.616} C_VEL
LIN {X 0,Y 509.812,Z 223.475,A -85,B 0,C 180,E1 -5452.658,E2 -5452.658} C_VEL
LIN {X 0,Y 509.856,Z 223.476,A -85,B 0,C 180,E1 -5455.801,E2 -5455.801} C_VEL
LIN {X 0,Y 509.861,Z 223.47,A -85,B 0,C 180,E1 -5458.721,E2 -5458.721} C_VEL
LIN {X 0,Y 509.866,Z 223.47,A -85,B 0,C 180,E1 -5461.154,E2 -5461.154} C_VEL
LIN {X 0,Y 509.88,Z 223.474,A -85,B 0,C 180,E1 -5463.826,E2 -5463.826} C_VEL
LIN {X 0,Y 509.896,Z 223.68,A -85,B 0,C 180,E1 -5466.223,E2 -5466.223} C_VEL
LIN {X 0,Y 511.32,Z 232.014,A -85,B 0,C 180,E1 -5467.79,E2 -5467.79} C_VEL
LIN {X 0,Y 510.867,Z 248.903,A -85,B 0,C 180,E1 -5470.72,E2 -5470.72} C_VEL
LIN {X 0,Y 510.386,Z 265.794,A -85,B 0,C 180,E1 -5473.602,E2 -5473.602} C_VEL
LIN {X 0,Y 510.284,Z 270.668,A -85,B 0,C 180,E1 -5474.396,E2 -5474.396} C_VEL
LIN {X 0,Y 511.459,Z 277.838,A -85,B 0,C 180,E1 -5474.568,E2 -5474.568} C_VEL
LIN {X 0,Y 512.215,Z 283.877,A -85,B 0,C 180,E1 -5474.679,E2 -5474.679} C_VEL
LIN {X 0,Y 511.726,Z 378.15,A -85,B 0,C 180,E1 -5476.041,E2 -5476.041} C_VEL
LIN {X 0,Y 511.446,Z 391.477,A -85,B 0,C 180,E1 -5476.388,E2 -5476.388} C_VEL
LIN {X 0,Y 511.154,Z 404.239,A -85,B 0,C 180,E1 -5476.886,E2 -5476.886} C_VEL
LIN {X 0,Y 510.862,Z 416.023,A -85,B 0,C 180,E1 -5477.513,E2 -5477.513} C_VEL
LIN {X 0,Y 510.586,Z 427.275,A -85,B 0,C 180,E1 -5478.285,E2 -5478.285} C_VEL
LIN {X 0,Y 510.208,Z 437.782,A -85,B 0,C 180,E1 -5479.181,E2 -5479.181} C_VEL
LIN {X 0,Y 509.944,Z 446.371,A -85,B 0,C 180,E1 -5480.079,E2 -5480.079} C_VEL
LIN {X 0,Y 509.681,Z 454.288,A -85,B 0,C 180,E1 -5481.075,E2 -5481.075} C_VEL
LIN {X 0,Y 509.508,Z 462.021,A -85,B 0,C 180,E1 -5482.27,E2 -5482.27} C_VEL
LIN {X 0,Y 509.318,Z 469.132,A -85,B 0,C 180,E1 -5483.661,E2 -5483.661} C_VEL
LIN {X 0,Y 509.249,Z 473.864,A -85,B 0,C 180,E1 -5484.852,E2 -5484.852} C_VEL
LIN {X 0,Y 509.248,Z 477.479,A -85,B 0,C 180,E1 -5486.042,E2 -5486.042} C_VEL
LIN {X 0,Y 509.203,Z 479.344,A -85,B 0,C 180,E1 -5486.834,E2 -5486.834} C_VEL
LIN {X 0,Y 509.163,Z 480.742,A -85,B 0,C 180,E1 -5487.625,E2 -5487.625} C_VEL
LIN {X 0,Y 509.075,Z 482.345,A -85,B 0,C 180,E1 -5489.208,E2 -5489.208} C_VEL
LIN {X 0,Y 509.067,Z 482.561,A -85,B 0,C 180,E1 -5489.999,E2 -5489.999} C_VEL
LIN {X 0,Y 509.114,Z 481.737,A -85,B 0,C 180,E1 -5491.581,E2 -5491.581} C_VEL
LIN {X 0,Y 509.163,Z 480.74,A -85,B 0,C 180,E1 -5492.372,E2 -5492.372} C_VEL
LIN {X 0,Y 509.203,Z 479.341,A -85,B 0,C 180,E1 -5493.163,E2 -5493.163} C_VEL
LIN {X 0,Y 509.206,Z 476.4,A -85,B 0,C 180,E1 -5494.352,E2 -5494.352} C_VEL
LIN {X 0,Y 509.311,Z 472.418,A -85,B 0,C 180,E1 -5495.542,E2 -5495.542} C_VEL
LIN {X 0,Y 509.368,Z 466.39,A -85,B 0,C 180,E1 -5496.913,E2 -5496.913} C_VEL
LIN {X 0,Y 509.562,Z 459.589,A -85,B 0,C 180,E1 -5498.126,E2 -5498.126} C_VEL
LIN {X 0,Y 509.764,Z 451.272,A -85,B 0,C 180,E1 -5499.321,E2 -5499.321} C_VEL
LIN {X 0,Y 510.014,Z 442.728,A -85,B 0,C 180,E1 -5500.318,E2 -5500.318} C_VEL
LIN {X 0,Y 510.386,Z 432.172,A -85,B 0,C 180,E1 -5501.315,E2 -5501.315} C_VEL
LIN {X 0,Y 510.69,Z 421.024,A -85,B 0,C 180,E1 -5502.162,E2 -5502.162} C_VEL
LIN {X 0,Y 511.017,Z 410.218,A -85,B 0,C 180,E1 -5502.811,E2 -5502.811} C_VEL
LIN {X 0,Y 511.317,Z 398.309,A -85,B 0,C 180,E1 -5503.359,E2 -5503.359} C_VEL
LIN {X 0,Y 511.599,Z 384.559,A -85,B 0,C 180,E1 -5503.807,E2 -5503.807} C_VEL
LIN {X 0,Y 511.749,Z 372.078,A -85,B 0,C 180,E1 -5504.057,E2 -5504.057} C_VEL
LIN {X 0,Y 512.163,Z 282.295,A -85,B 0,C 180,E1 -5505.343,E2 -5505.343} C_VEL
LIN {X 0,Y 510.276,Z 270.614,A -85,B 0,C 180,E1 -5505.589,E2 -5505.589} C_VEL
LIN {X 0,Y 510.668,Z 253.239,A -85,B 0,C 180,E1 -5508.452,E2 -5508.452} C_VEL
LIN {X 0,Y 511.166,Z 234.773,A -85,B 0,C 180,E1 -5511.577,E2 -5511.577} C_VEL
LIN {X 0,Y 511.028,Z 229.822,A -85,B 0,C 180,E1 -5512.433,E2 -5512.433} C_VEL
LIN {X 0,Y 509.881,Z 223.576,A -85,B 0,C 180,E1 -5513.613,E2 -5513.613} C_VEL
LIN {X 0,Y 509.881,Z 223.471,A -85,B 0,C 180,E1 -5517.054,E2 -5517.054} C_VEL
LIN {X 0,Y 509.862,Z 223.478,A -85,B 0,C 180,E1 -5519.749,E2 -5519.749} C_VEL
LIN {X 0,Y 509.877,Z 223.469,A -85,B 0,C 180,E1 -5522.771,E2 -5522.771} C_VEL
LIN {X 0,Y 509.826,Z 223.479,A -85,B 0,C 180,E1 -5525.575,E2 -5525.575} C_VEL
LIN {X 0,Y 509.85,Z 223.476,A -85,B 0,C 180,E1 -5528.336,E2 -5528.336} C_VEL
LIN {X 0,Y 509.833,Z 223.474,A -85,B 0,C 180,E1 -5531.425,E2 -5531.425} C_VEL
LIN {X 0,Y 509.841,Z 223.474,A -85,B 0,C 180,E1 -5534.667,E2 -5534.667} C_VEL
LIN {X 0,Y 509.792,Z 223.479,A -85,B 0,C 180,E1 -5537.502,E2 -5537.502} C_VEL
LIN {X 0,Y 509.832,Z 223.477,A -85,B 0,C 180,E1 -5540.643,E2 -5540.643} C_VEL
LIN {X 0,Y 509.766,Z 223.481,A -85,B 0,C 180,E1 -5543.638,E2 -5543.638} C_VEL
LIN {X 0,Y 509.838,Z 223.478,A -85,B 0,C 180,E1 -5546.534,E2 -5546.534} C_VEL
LIN {X 0,Y 509.825,Z 223.473,A -85,B 0,C 180,E1 -5549.329,E2 -5549.329} C_VEL
LIN {X 0,Y 509.82,Z 223.477,A -85,B 0,C 180,E1 -5552.046,E2 -5552.046} C_VEL
LIN {X 0,Y 509.795,Z 223.485,A -85,B 0,C 180,E1 -5554.696,E2 -5554.696} C_VEL
LIN {X 0,Y 509.818,Z 223.474,A -85,B 0,C 180,E1 -5557.455,E2 -5557.455} C_VEL
LIN {X 0,Y 509.819,Z 223.481,A -85,B 0,C 180,E1 -5560.676,E2 -5560.676} C_VEL
LIN {X 0,Y 509.784,Z 223.483,A -85,B 0,C 180,E1 -5563.167,E2 -5563.167} C_VEL
LIN {X 0,Y 509.829,Z 223.474,A -85,B 0,C 180,E1 -5565.629,E2 -5565.629} C_VEL
LIN {X 0,Y 509.887,Z 223.471,A -85,B 0,C 180,E1 -5568.869,E2 -5568.869} C_VEL
LIN {X 0,Y 509.874,Z 223.467,A -85,B 0,C 180,E1 -5572.073,E2 -5572.073} C_VEL
LIN {X 0,Y 509.949,Z 223.458,A -85,B 0,C 180,E1 -5574.459,E2 -5574.459} C_VEL
LIN {X 0,Y 510.026,Z 223.452,A -85,B 0,C 180,E1 -5577.626,E2 -5577.626} C_VEL
LIN {X 0,Y 510.031,Z 223.448,A -85,B 0,C 180,E1 -5579.995,E2 -5579.995} C_VEL
LIN {X 0,Y 510.029,Z 223.448,A -85,B 0,C 180,E1 -5582.364,E2 -5582.364} C_VEL
LIN {X 0,Y 509.954,Z 223.466,A -85,B 0,C 180,E1 -5585.53,E2 -5585.53} C_VEL
LIN {X 0,Y 509.89,Z 223.467,A -85,B 0,C 180,E1 -5588.715,E2 -5588.715} C_VEL
LIN {X 0,Y 509.923,Z 223.467,A -85,B 0,C 180,E1 -5591.925,E2 -5591.925} C_VEL
LIN {X 0,Y 509.862,Z 223.474,A -85,B 0,C 180,E1 -5595.236,E2 -5595.236} C_VEL
LIN {X 0,Y 509.855,Z 223.477,A -85,B 0,C 180,E1 -5597.996,E2 -5597.996} C_VEL
LIN {X 0,Y 509.825,Z 223.476,A -85,B 0,C 180,E1 -5600.996,E2 -5600.996} C_VEL
LIN {X 0,Y 509.834,Z 223.482,A -85,B 0,C 180,E1 -5603.556,E2 -5603.556} C_VEL
LIN {X 0,Y 509.937,Z 223.671,A -85,B 0,C 180,E1 -5604.712,E2 -5604.712} C_VEL
LIN {X 0,Y 510.62,Z 229.083,A -85,B 0,C 180,E1 -5605.686,E2 -5605.686} C_VEL
LIN {X 0,Y 510.315,Z 247.417,A -85,B 0,C 180,E1 -5608.809,E2 -5608.809} C_VEL
LIN {X 0,Y 510.245,Z 256.97,A -85,B 0,C 180,E1 -5610.431,E2 -5610.431} C_VEL
LIN {X 0,Y 510.469,Z 258.738,A -85,B 0,C 180,E1 -5610.502,E2 -5610.502} C_VEL
LIN {X 0,Y 512.193,Z 268.63,A -85,B 0,C 180,E1 -5610.702,E2 -5610.702} C_VEL
LIN {X 0,Y 511.69,Z 364.869,A -85,B 0,C 180,E1 -5612.1,E2 -5612.1} C_VEL
LIN {X 0,Y 511.464,Z 378.693,A -85,B 0,C 180,E1 -5612.471,E2 -5612.471} C_VEL
LIN {X 0,Y 511.256,Z 390.295,A -85,B 0,C 180,E1 -5612.932,E2 -5612.932} C_VEL
LIN {X 0,Y 510.955,Z 401.955,A -85,B 0,C 180,E1 -5613.548,E2 -5613.548} C_VEL
LIN {X 0,Y 510.572,Z 413.622,A -85,B 0,C 180,E1 -5614.349,E2 -5614.349} C_VEL
LIN {X 0,Y 510.279,Z 423.76,A -85,B 0,C 180,E1 -5615.218,E2 -5615.218} C_VEL
LIN {X 0,Y 509.452,Z 428.216,A -85,B 0,C 180,E1 -5615.646,E2 -5615.646} C_VEL
LIN {X 0,Y 506.386,Z 435.14,A -85,B 0,C 180,E1 -5616.369,E2 -5616.369} C_VEL
LIN {X 0,Y 503.338,Z 441.485,A -85,B 0,C 180,E1 -5617.163,E2 -5617.163} C_VEL
LIN {X 0,Y 502.548,Z 445.031,A -85,B 0,C 180,E1 -5617.694,E2 -5617.694} C_VEL
LIN {X 0,Y 502.355,Z 452.346,A -85,B 0,C 180,E1 -5619.007,E2 -5619.007} C_VEL
LIN {X 0,Y 502.207,Z 457.052,A -85,B 0,C 180,E1 -5620.061,E2 -5620.061} C_VEL
LIN {X 0,Y 502.168,Z 460.882,A -85,B 0,C 180,E1 -5621.12,E2 -5621.12} C_VEL
LIN {X 0,Y 502.061,Z 463.954,A -85,B 0,C 180,E1 -5622.205,E2 -5622.205} C_VEL
LIN {X 0,Y 502.004,Z 466.217,A -85,B 0,C 180,E1 -5623.303,E2 -5623.303} C_VEL
LIN {X 0,Y 502.011,Z 467.738,A -85,B 0,C 180,E1 -5624.443,E2 -5624.443} C_VEL
LIN {X 0,Y 501.983,Z 468.47,A -85,B 0,C 180,E1 -5625.574,E2 -5625.574} C_VEL
LIN {X 0,Y 501.974,Z 468.409,A -85,B 0,C 180,E1 -5626.71,E2 -5626.71} C_VEL
LIN {X 0,Y 502.003,Z 467.486,A -85,B 0,C 180,E1 -5627.889,E2 -5627.889} C_VEL
LIN {X 0,Y 502.043,Z 465.644,A -85,B 0,C 180,E1 -5629.094,E2 -5629.094} C_VEL
LIN {X 0,Y 502.097,Z 462.775,A -85,B 0,C 180,E1 -5630.327,E2 -5630.327} C_VEL
LIN {X 0,Y 502.19,Z 458.735,A -85,B 0,C 180,E1 -5631.587,E2 -5631.587} C_VEL
LIN {X 0,Y 502.349,Z 452.638,A -85,B 0,C 180,E1 -5633.019,E2 -5633.019} C_VEL
LIN {X 0,Y 502.529,Z 446.239,A -85,B 0,C 180,E1 -5634.193,E2 -5634.193} C_VEL
LIN {X 0,Y 502.763,Z 438.695,A -85,B 0,C 180,E1 -5635.321,E2 -5635.321} C_VEL
LIN {X 0,Y 503.062,Z 430.012,A -85,B 0,C 180,E1 -5636.383,E2 -5636.383} C_VEL
LIN {X 0,Y 503.372,Z 420.111,A -85,B 0,C 180,E1 -5637.368,E2 -5637.368} C_VEL
LIN {X 0,Y 503.712,Z 410.028,A -85,B 0,C 180,E1 -5638.178,E2 -5638.178} C_VEL
LIN {X 0,Y 504.068,Z 398.023,A -85,B 0,C 180,E1 -5638.946,E2 -5638.946} C_VEL
LIN {X 0,Y 504.453,Z 385.83,A -85,B 0,C 180,E1 -5639.54,E2 -5639.54} C_VEL
LIN {X 0,Y 504.681,Z 372.914,A -85,B 0,C 180,E1 -5639.987,E2 -5639.987} C_VEL
LIN {X 0,Y 504.851,Z 359.943,A -85,B 0,C 180,E1 -5640.271,E2 -5640.271} C_VEL
LIN {X 0,Y 505.222,Z 268.611,A -85,B 0,C 180,E1 -5641.605,E2 -5641.605} C_VEL
LIN {X 0,Y 503.364,Z 258.172,A -85,B 0,C 180,E1 -5641.832,E2 -5641.832} C_VEL
LIN {X 0,Y 503.298,Z 257.435,A -85,B 0,C 180,E1 -5641.885,E2 -5641.885} C_VEL
LIN {X 0,Y 503.813,Z 240.723,A -85,B 0,C 180,E1 -5645.035,E2 -5645.035} C_VEL
LIN {X 0,Y 503.986,Z 230.787,A -85,B 0,C 180,E1 -5646.956,E2 -5646.956} C_VEL
LIN {X 0,Y 502.813,Z 224.402,A -85,B 0,C 180,E1 -5648.315,E2 -5648.315} C_VEL
LIN {X 0,Y 502.754,Z 224.358,A -85,B 0,C 180,E1 -5651.247,E2 -5651.247} C_VEL
LIN {X 0,Y 502.754,Z 224.356,A -85,B 0,C 180,E1 -5653.767,E2 -5653.767} C_VEL
LIN {X 0,Y 502.776,Z 224.356,A -85,B 0,C 180,E1 -5656.255,E2 -5656.255} C_VEL
LIN {X 0,Y 502.824,Z 224.353,A -85,B 0,C 180,E1 -5658.717,E2 -5658.717} C_VEL
LIN {X 0,Y 502.828,Z 224.345,A -85,B 0,C 180,E1 -5661.967,E2 -5661.967} C_VEL
LIN {X 0,Y 502.889,Z 224.34,A -85,B 0,C 180,E1 -5664.387,E2 -5664.387} C_VEL
LIN {X 0,Y 502.951,Z 224.33,A -85,B 0,C 180,E1 -5667.599,E2 -5667.599} C_VEL
LIN {X 0,Y 502.944,Z 224.33,A -85,B 0,C 180,E1 -5670.001,E2 -5670.001} C_VEL
LIN {X 0,Y 502.951,Z 224.33,A -85,B 0,C 180,E1 -5672.404,E2 -5672.404} C_VEL
LIN {X 0,Y 502.89,Z 224.34,A -85,B 0,C 180,E1 -5675.615,E2 -5675.615} C_VEL
LIN {X 0,Y 502.827,Z 224.348,A -85,B 0,C 180,E1 -5678.845,E2 -5678.845} C_VEL
LIN {X 0,Y 502.822,Z 224.346,A -85,B 0,C 180,E1 -5682.103,E2 -5682.103} C_VEL
LIN {X 0,Y 502.778,Z 224.358,A -85,B 0,C 180,E1 -5685.403,E2 -5685.403} C_VEL
LIN {X 0,Y 502.774,Z 224.354,A -85,B 0,C 180,E1 -5688.126,E2 -5688.126} C_VEL
LIN {X 0,Y 502.759,Z 224.353,A -85,B 0,C 180,E1 -5690.54,E2 -5690.54} C_VEL
LIN {X 0,Y 502.735,Z 224.357,A -85,B 0,C 180,E1 -5693.044,E2 -5693.044} C_VEL
LIN {X 0,Y 502.782,Z 224.357,A -85,B 0,C 180,E1 -5695.68,E2 -5695.68} C_VEL
LIN {X 0,Y 502.78,Z 224.354,A -85,B 0,C 180,E1 -5698.377,E2 -5698.377} C_VEL
LIN {X 0,Y 502.744,Z 224.357,A -85,B 0,C 180,E1 -5701.506,E2 -5701.506} C_VEL
LIN {X 0,Y 502.75,Z 224.36,A -85,B 0,C 180,E1 -5704.45,E2 -5704.45} C_VEL
LIN {X 0,Y 502.727,Z 224.357,A -85,B 0,C 180,E1 -5707.184,E2 -5707.184} C_VEL
LIN {X 0,Y 502.771,Z 224.356,A -85,B 0,C 180,E1 -5710.018,E2 -5710.018} C_VEL
LIN {X 0,Y 502.778,Z 224.357,A -85,B 0,C 180,E1 -5712.208,E2 -5712.208} C_VEL
LIN {X 0,Y 502.756,Z 224.354,A -85,B 0,C 180,E1 -5715.475,E2 -5715.475} C_VEL
LIN {X 0,Y 502.797,Z 224.349,A -85,B 0,C 180,E1 -5717.872,E2 -5717.872} C_VEL
LIN {X 0,Y 502.782,Z 224.355,A -85,B 0,C 180,E1 -5721.032,E2 -5721.032} C_VEL
LIN {X 0,Y 502.75,Z 224.355,A -85,B 0,C 180,E1 -5724.174,E2 -5724.174} C_VEL
LIN {X 0,Y 502.8,Z 224.357,A -85,B 0,C 180,E1 -5727,E2 -5727} C_VEL
LIN {X 0,Y 502.788,Z 224.349,A -85,B 0,C 180,E1 -5730.072,E2 -5730.072} C_VEL
LIN {X 0,Y 502.806,Z 224.349,A -85,B 0,C 180,E1 -5732.54,E2 -5732.54} C_VEL
LIN {X 0,Y 502.806,Z 224.356,A -85,B 0,C 180,E1 -5735.306,E2 -5735.306} C_VEL
LIN {X 0,Y 502.763,Z 224.355,A -85,B 0,C 180,E1 -5737.833,E2 -5737.833} C_VEL
LIN {X 0,Y 502.808,Z 224.347,A -85,B 0,C 180,E1 -5740.407,E2 -5740.407} C_VEL
LIN {X 0,Y 502.806,Z 224.349,A -85,B 0,C 180,E1 -5742.937,E2 -5742.937} C_VEL
LIN {X 0,Y 502.834,Z 224.351,A -85,B 0,C 180,E1 -5745.435,E2 -5745.435} C_VEL
LIN {X 0,Y 502.871,Z 224.339,A -85,B 0,C 180,E1 -5748.723,E2 -5748.723} C_VEL
LIN {X 0,Y 502.878,Z 224.345,A -85,B 0,C 180,E1 -5751.972,E2 -5751.972} C_VEL
LIN {X 0,Y 502.906,Z 224.337,A -85,B 0,C 180,E1 -5754.392,E2 -5754.392} C_VEL
LIN {X 0,Y 503.019,Z 224.325,A -85,B 0,C 180,E1 -5757.603,E2 -5757.603} C_VEL
LIN {X 0,Y 502.975,Z 224.327,A -85,B 0,C 180,E1 -5760.806,E2 -5760.806} C_VEL
LIN {X 0,Y 503.015,Z 224.327,A -85,B 0,C 180,E1 -5762.407,E2 -5762.407} C_VEL
LIN {X 0,Y 502.911,Z 224.335,A -85,B 0,C 180,E1 -5765.619,E2 -5765.619} C_VEL
LIN {X 0,Y 502.858,Z 224.346,A -85,B 0,C 180,E1 -5768.039,E2 -5768.039} C_VEL
LIN {X 0,Y 502.885,Z 224.338,A -85,B 0,C 180,E1 -5771.288,E2 -5771.288} C_VEL
LIN {X 0,Y 502.841,Z 224.353,A -85,B 0,C 180,E1 -5774.575,E2 -5774.575} C_VEL
LIN {X 0,Y 502.824,Z 224.348,A -85,B 0,C 180,E1 -5777.073,E2 -5777.073} C_VEL
LIN {X 0,Y 502.827,Z 224.345,A -85,B 0,C 180,E1 -5779.604,E2 -5779.604} C_VEL
LIN {X 0,Y 502.819,Z 224.353,A -85,B 0,C 180,E1 -5782.705,E2 -5782.705} C_VEL
LIN {X 0,Y 502.794,Z 224.349,A -85,B 0,C 180,E1 -5785.682,E2 -5785.682} C_VEL
LIN {X 0,Y 502.791,Z 224.35,A -85,B 0,C 180,E1 -5788.38,E2 -5788.38} C_VEL
LIN {X 0,Y 502.805,Z 224.357,A -85,B 0,C 180,E1 -5791.146,E2 -5791.146} C_VEL
LIN {X 0,Y 502.803,Z 224.348,A -85,B 0,C 180,E1 -5793.998,E2 -5793.998} C_VEL
LIN {X 0,Y 502.781,Z 224.358,A -85,B 0,C 180,E1 -5797.177,E2 -5797.177} C_VEL
LIN {X 0,Y 502.79,Z 224.351,A -85,B 0,C 180,E1 -5800.019,E2 -5800.019} C_VEL
LIN {X 0,Y 502.757,Z 224.358,A -85,B 0,C 180,E1 -5803.236,E2 -5803.236} C_VEL
LIN {X 0,Y 502.786,Z 224.359,A -85,B 0,C 180,E1 -5805.66,E2 -5805.66} C_VEL
LIN {X 0,Y 502.782,Z 224.351,A -85,B 0,C 180,E1 -5809.013,E2 -5809.013} C_VEL
LIN {X 0,Y 502.782,Z 224.357,A -85,B 0,C 180,E1 -5812.044,E2 -5812.044} C_VEL
LIN {X 0,Y 502.807,Z 224.347,A -85,B 0,C 180,E1 -5815.034,E2 -5815.034} C_VEL
LIN {X 0,Y 502.798,Z 224.356,A -85,B 0,C 180,E1 -5817.915,E2 -5817.915} C_VEL
LIN {X 0,Y 502.829,Z 224.349,A -85,B 0,C 180,E1 -5820.711,E2 -5820.711} C_VEL
LIN {X 0,Y 502.84,Z 224.348,A -85,B 0,C 180,E1 -5823.449,E2 -5823.449} C_VEL
LIN {X 0,Y 502.857,Z 224.391,A -85,B 0,C 180,E1 -5825.979,E2 -5825.979} C_VEL
LIN {X 0,Y 503.584,Z 228.302,A -85,B 0,C 180,E1 -5826.779,E2 -5826.779} C_VEL
LIN {X 0,Y 504.399,Z 234.353,A -85,B 0,C 180,E1 -5827.9,E2 -5827.9} C_VEL
LIN {X 0,Y 503.777,Z 252.439,A -85,B 0,C 180,E1 -5831.073,E2 -5831.073} C_VEL
LIN {X 0,Y 503.311,Z 269.255,A -85,B 0,C 180,E1 -5833.979,E2 -5833.979} C_VEL
LIN {X 0,Y 503.328,Z 270.998,A -85,B 0,C 180,E1 -5834.199,E2 -5834.199} C_VEL
LIN {X 0,Y 505.366,Z 283.98,A -85,B 0,C 180,E1 -5834.47,E2 -5834.47} C_VEL
LIN {X 0,Y 504.828,Z 378.994,A -85,B 0,C 180,E1 -5835.872,E2 -5835.872} C_VEL
LIN {X 0,Y 504.526,Z 392.76,A -85,B 0,C 180,E1 -5836.249,E2 -5836.249} C_VEL
LIN {X 0,Y 504.195,Z 405.137,A -85,B 0,C 180,E1 -5836.753,E2 -5836.753} C_VEL
LIN {X 0,Y 503.841,Z 417.6,A -85,B 0,C 180,E1 -5837.449,E2 -5837.449} C_VEL
LIN {X 0,Y 503.572,Z 428.413,A -85,B 0,C 180,E1 -5838.221,E2 -5838.221} C_VEL
LIN {X 0,Y 503.174,Z 438.701,A -85,B 0,C 180,E1 -5839.13,E2 -5839.13} C_VEL
LIN {X 0,Y 502.867,Z 447.936,A -85,B 0,C 180,E1 -5840.141,E2 -5840.141} C_VEL
LIN {X 0,Y 502.595,Z 456.916,A -85,B 0,C 180,E1 -5841.353,E2 -5841.353} C_VEL
LIN {X 0,Y 502.364,Z 464.145,A -85,B 0,C 180,E1 -5842.563,E2 -5842.563} C_VEL
LIN {X 0,Y 502.246,Z 469.02,A -85,B 0,C 180,E1 -5843.571,E2 -5843.571} C_VEL
LIN {X 0,Y 502.183,Z 473.758,A -85,B 0,C 180,E1 -5844.779,E2 -5844.779} C_VEL
LIN {X 0,Y 502.141,Z 477.376,A -85,B 0,C 180,E1 -5845.986,E2 -5845.986} C_VEL
LIN {X 0,Y 502.124,Z 479.243,A -85,B 0,C 180,E1 -5846.789,E2 -5846.789} C_VEL
LIN {X 0,Y 502.068,Z 480.642,A -85,B 0,C 180,E1 -5847.592,E2 -5847.592} C_VEL
LIN {X 0,Y 502.038,Z 481.639,A -85,B 0,C 180,E1 -5848.394,E2 -5848.394} C_VEL
LIN {X 0,Y 501.982,Z 482.463,A -85,B 0,C 180,E1 -5849.999,E2 -5849.999} C_VEL
LIN {X 0,Y 502.038,Z 481.637,A -85,B 0,C 180,E1 -5851.603,E2 -5851.603} C_VEL
LIN {X 0,Y 502.068,Z 480.638,A -85,B 0,C 180,E1 -5852.405,E2 -5852.405} C_VEL
LIN {X 0,Y 502.123,Z 479.237,A -85,B 0,C 180,E1 -5853.208,E2 -5853.208} C_VEL
LIN {X 0,Y 502.104,Z 476.292,A -85,B 0,C 180,E1 -5854.414,E2 -5854.414} C_VEL
LIN {X 0,Y 502.228,Z 472.306,A -85,B 0,C 180,E1 -5855.62,E2 -5855.62} C_VEL
LIN {X 0,Y 502.294,Z 466.268,A -85,B 0,C 180,E1 -5857.011,E2 -5857.011} C_VEL
LIN {X 0,Y 502.488,Z 459.459,A -85,B 0,C 180,E1 -5858.241,E2 -5858.241} C_VEL
LIN {X 0,Y 502.737,Z 451.134,A -85,B 0,C 180,E1 -5859.453,E2 -5859.453} C_VEL
LIN {X 0,Y 502.99,Z 442.576,A -85,B 0,C 180,E1 -5860.464,E2 -5860.464} C_VEL
LIN {X 0,Y 503.41,Z 432.006,A -85,B 0,C 180,E1 -5861.473,E2 -5861.473} C_VEL
LIN {X 0,Y 503.716,Z 420.847,A -85,B 0,C 180,E1 -5862.333,E2 -5862.333} C_VEL
LIN {X 0,Y 504.066,Z 410.022,A -85,B 0,C 180,E1 -5862.991,E2 -5862.991} C_VEL
LIN {X 0,Y 504.415,Z 398.088,A -85,B 0,C 180,E1 -5863.546,E2 -5863.546} C_VEL
LIN {X 0,Y 504.724,Z 384.305,A -85,B 0,C 180,E1 -5863.999,E2 -5863.999} C_VEL
LIN {X 0,Y 504.864,Z 371.713,A -85,B 0,C 180,E1 -5864.252,E2 -5864.252} C_VEL
LIN {X 0,Y 505.342,Z 283.342,A -85,B 0,C 180,E1 -5865.539,E2 -5865.539} C_VEL
LIN {X 0,Y 503.263,Z 270.383,A -85,B 0,C 180,E1 -5865.821,E2 -5865.821} C_VEL
LIN {X 0,Y 503.736,Z 251.894,A -85,B 0,C 180,E1 -5868.926,E2 -5868.926} C_VEL
LIN {X 0,Y 504.214,Z 234.644,A -85,B 0,C 180,E1 -5871.89,E2 -5871.89} C_VEL
LIN {X 0,Y 504.037,Z 230.976,A -85,B 0,C 180,E1 -5872.539,E2 -5872.539} C_VEL
LIN {X 0,Y 502.859,Z 224.535,A -85,B 0,C 180,E1 -5873.744,E2 -5873.744} C_VEL
LIN {X 0,Y 502.843,Z 224.347,A -85,B 0,C 180,E1 -5876.565,E2 -5876.565} C_VEL
LIN {X 0,Y 502.827,Z 224.35,A -85,B 0,C 180,E1 -5879.286,E2 -5879.286} C_VEL
LIN {X 0,Y 502.787,Z 224.358,A -85,B 0,C 180,E1 -5882.082,E2 -5882.082} C_VEL
LIN {X 0,Y 502.801,Z 224.35,A -85,B 0,C 180,E1 -5884.963,E2 -5884.963} C_VEL
LIN {X 0,Y 502.793,Z 224.353,A -85,B 0,C 180,E1 -5888.482,E2 -5888.482} C_VEL
LIN {X 0,Y 502.774,Z 224.352,A -85,B 0,C 180,E1 -5891.068,E2 -5891.068} C_VEL
LIN {X 0,Y 502.787,Z 224.354,A -85,B 0,C 180,E1 -5894.527,E2 -5894.527} C_VEL
LIN {X 0,Y 502.767,Z 224.357,A -85,B 0,C 180,E1 -5897.854,E2 -5897.854} C_VEL
LIN {X 0,Y 502.783,Z 224.352,A -85,B 0,C 180,E1 -5901.019,E2 -5901.019} C_VEL
LIN {X 0,Y 502.75,Z 224.36,A -85,B 0,C 180,E1 -5904.17,E2 -5904.17} C_VEL
LIN {X 0,Y 502.802,Z 224.35,A -85,B 0,C 180,E1 -5906.995,E2 -5906.995} C_VEL
LIN {X 0,Y 502.807,Z 224.35,A -85,B 0,C 180,E1 -5910.063,E2 -5910.063} C_VEL
LIN {X 0,Y 502.77,Z 224.35,A -85,B 0,C 180,E1 -5913.456,E2 -5913.456} C_VEL
LIN {X 0,Y 502.754,Z 224.356,A -85,B 0,C 180,E1 -5916.08,E2 -5916.08} C_VEL
LIN {X 0,Y 502.756,Z 224.361,A -85,B 0,C 180,E1 -5918.684,E2 -5918.684} C_VEL
LIN {X 0,Y 502.785,Z 224.35,A -85,B 0,C 180,E1 -5921.893,E2 -5921.893} C_VEL
LIN {X 0,Y 502.812,Z 224.35,A -85,B 0,C 180,E1 -5925.424,E2 -5925.424} C_VEL
LIN {X 0,Y 502.855,Z 224.345,A -85,B 0,C 180,E1 -5928.712,E2 -5928.712} C_VEL
LIN {X 0,Y 502.842,Z 224.344,A -85,B 0,C 180,E1 -5931.961,E2 -5931.961} C_VEL
LIN {X 0,Y 502.904,Z 224.335,A -85,B 0,C 180,E1 -5934.381,E2 -5934.381} C_VEL
LIN {X 0,Y 502.996,Z 224.329,A -85,B 0,C 180,E1 -5937.593,E2 -5937.593} C_VEL
LIN {X 0,Y 503.003,Z 224.324,A -85,B 0,C 180,E1 -5939.995,E2 -5939.995} C_VEL
LIN {X 0,Y 503,Z 224.324,A -85,B 0,C 180,E1 -5942.397,E2 -5942.397} C_VEL
LIN {X 0,Y 502.907,Z 224.343,A -85,B 0,C 180,E1 -5945.608,E2 -5945.608} C_VEL
LIN {X 0,Y 502.849,Z 224.345,A -85,B 0,C 180,E1 -5948.838,E2 -5948.838} C_VEL
LIN {X 0,Y 502.866,Z 224.344,A -85,B 0,C 180,E1 -5952.095,E2 -5952.095} C_VEL
LIN {X 0,Y 502.817,Z 224.354,A -85,B 0,C 180,E1 -5955.394,E2 -5955.394} C_VEL
LIN {X 0,Y 502.812,Z 224.353,A -85,B 0,C 180,E1 -5958.117,E2 -5958.117} C_VEL
LIN {X 0,Y 502.765,Z 224.358,A -85,B 0,C 180,E1 -5961.305,E2 -5961.305} C_VEL
LIN {X 0,Y 502.903,Z 224.507,A -85,B 0,C 180,E1 -5964.555,E2 -5964.555} C_VEL
LIN {X 0,Y 503.667,Z 230.306,A -85,B 0,C 180,E1 -5965.623,E2 -5965.623} C_VEL
LIN {X 0,Y 503.321,Z 248.75,A -85,B 0,C 180,E1 -5968.79,E2 -5968.79} C_VEL
LIN {X 0,Y 503.25,Z 257.151,A -85,B 0,C 180,E1 -5970.219,E2 -5970.219} C_VEL
LIN {X 0,Y 504.176,Z 262.752,A -85,B 0,C 180,E1 -5970.36,E2 -5970.36} C_VEL
LIN {X 0,Y 505.39,Z 270.479,A -85,B 0,C 180,E1 -5970.515,E2 -5970.515} C_VEL
LIN {X 0,Y 504.797,Z 365.095,A -85,B 0,C 180,E1 -5971.913,E2 -5971.913} C_VEL
LIN {X 0,Y 504.576,Z 378.804,A -85,B 0,C 180,E1 -5972.287,E2 -5972.287} C_VEL
LIN {X 0,Y 504.305,Z 391.321,A -85,B 0,C 180,E1 -5972.795,E2 -5972.795} C_VEL
LIN {X 0,Y 503.991,Z 402.806,A -85,B 0,C 180,E1 -5973.426,E2 -5973.426} C_VEL
LIN {X 0,Y 503.588,Z 414.524,A -85,B 0,C 180,E1 -5974.252,E2 -5974.252} C_VEL
LIN {X 0,Y 503.238,Z 424.865,A -85,B 0,C 180,E1 -5975.166,E2 -5975.166} C_VEL
LIN {X 0,Y 502.909,Z 434.116,A -85,B 0,C 180,E1 -5976.178,E2 -5976.178} C_VEL
LIN {X 0,Y 502.625,Z 442.599,A -85,B 0,C 180,E1 -5977.319,E2 -5977.319} C_VEL
LIN {X 0,Y 502.548,Z 445.031,A -85,B 0,C 180,E1 -5977.694,E2 -5977.694} C_VEL
LIN {X 0,Y 501.763,Z 448.389,A -85,B 0,C 180,E1 -5978.244,E2 -5978.244} C_VEL
LIN {X 0,Y 498.754,Z 453.431,A -85,B 0,C 180,E1 -5979.161,E2 -5979.161} C_VEL
LIN {X 0,Y 495.791,Z 457.788,A -85,B 0,C 180,E1 -5980.131,E2 -5980.131} C_VEL
LIN {X 0,Y 495.086,Z 460.024,A -85,B 0,C 180,E1 -5980.76,E2 -5980.76} C_VEL
LIN {X 0,Y 495.019,Z 463.264,A -85,B 0,C 180,E1 -5981.847,E2 -5981.847} C_VEL
LIN {X 0,Y 494.933,Z 465.765,A -85,B 0,C 180,E1 -5982.957,E2 -5982.957} C_VEL
LIN {X 0,Y 494.92,Z 467.5,A -85,B 0,C 180,E1 -5984.081,E2 -5984.081} C_VEL
LIN {X 0,Y 494.916,Z 468.438,A -85,B 0,C 180,E1 -5985.225,E2 -5985.225} C_VEL
LIN {X 0,Y 494.868,Z 468.591,A -85,B 0,C 180,E1 -5986.398,E2 -5986.398} C_VEL
LIN {X 0,Y 494.909,Z 467.912,A -85,B 0,C 180,E1 -5987.586,E2 -5987.586} C_VEL
LIN {X 0,Y 494.947,Z 465.587,A -85,B 0,C 180,E1 -5989.221,E2 -5989.221} C_VEL
LIN {X 0,Y 495.026,Z 463.108,A -85,B 0,C 180,E1 -5990.294,E2 -5990.294} C_VEL
LIN {X 0,Y 495.142,Z 458.064,A -85,B 0,C 180,E1 -5991.873,E2 -5991.873} C_VEL
LIN {X 0,Y 495.277,Z 453.202,A -85,B 0,C 180,E1 -5993.02,E2 -5993.02} C_VEL
LIN {X 0,Y 495.465,Z 446.987,A -85,B 0,C 180,E1 -5994.198,E2 -5994.198} C_VEL
LIN {X 0,Y 495.72,Z 438.751,A -85,B 0,C 180,E1 -5995.454,E2 -5995.454} C_VEL
LIN {X 0,Y 496.059,Z 429.403,A -85,B 0,C 180,E1 -5996.605,E2 -5996.605} C_VEL
LIN {X 0,Y 496.46,Z 418.936,A -85,B 0,C 180,E1 -5997.633,E2 -5997.633} C_VEL
LIN {X 0,Y 496.783,Z 408.805,A -85,B 0,C 180,E1 -5998.439,E2 -5998.439} C_VEL
LIN {X 0,Y 497.178,Z 397.168,A -85,B 0,C 180,E1 -5999.177,E2 -5999.177} C_VEL
LIN {X 0,Y 497.543,Z 384.293,A -85,B 0,C 180,E1 -5999.789,E2 -5999.789} C_VEL
LIN {X 0,Y 497.823,Z 371.06,A -85,B 0,C 180,E1 -6000.231,E2 -6000.231} C_VEL
LIN {X 0,Y 497.999,Z 357.238,A -85,B 0,C 180,E1 -6000.508,E2 -6000.508} C_VEL
LIN {X 0,Y 498.417,Z 269.74,A -85,B 0,C 180,E1 -6001.802,E2 -6001.802} C_VEL
LIN {X 0,Y 496.35,Z 258.105,A -85,B 0,C 180,E1 -6002.062,E2 -6002.062} C_VEL
LIN {X 0,Y 496.311,Z 257.319,A -85,B 0,C 180,E1 -6002.143,E2 -6002.143} C_VEL
LIN {X 0,Y 496.854,Z 241.798,A -85,B 0,C 180,E1 -6005.116,E2 -6005.116} C_VEL
LIN {X 0,Y 497.108,Z 233.422,A -85,B 0,C 180,E1 -6006.751,E2 -6006.751} C_VEL
LIN {X 0,Y 495.805,Z 225.588,A -85,B 0,C 180,E1 -6008.376,E2 -6008.376} C_VEL
LIN {X 0,Y 495.743,Z 225.235,A -85,B 0,C 180,E1 -6008.591,E2 -6008.591} C_VEL
LIN {X 0,Y 495.72,Z 225.236,A -85,B 0,C 180,E1 -6011.828,E2 -6011.828} C_VEL
LIN {X 0,Y 495.741,Z 225.228,A -85,B 0,C 180,E1 -6015.217,E2 -6015.217} C_VEL
LIN {X 0,Y 495.802,Z 225.229,A -85,B 0,C 180,E1 -6018.555,E2 -6018.555} C_VEL
LIN {X 0,Y 495.801,Z 225.22,A -85,B 0,C 180,E1 -6021.852,E2 -6021.852} C_VEL
LIN {X 0,Y 495.842,Z 225.217,A -85,B 0,C 180,E1 -6024.307,E2 -6024.307} C_VEL
LIN {X 0,Y 495.921,Z 225.206,A -85,B 0,C 180,E1 -6027.565,E2 -6027.565} C_VEL
LIN {X 0,Y 495.916,Z 225.206,A -85,B 0,C 180,E1 -6030.001,E2 -6030.001} C_VEL
LIN {X 0,Y 495.922,Z 225.206,A -85,B 0,C 180,E1 -6032.438,E2 -6032.438} C_VEL
LIN {X 0,Y 495.844,Z 225.217,A -85,B 0,C 180,E1 -6035.695,E2 -6035.695} C_VEL
LIN {X 0,Y 495.804,Z 225.22,A -85,B 0,C 180,E1 -6038.15,E2 -6038.15} C_VEL
LIN {X 0,Y 495.806,Z 225.228,A -85,B 0,C 180,E1 -6041.447,E2 -6041.447} C_VEL
LIN {X 0,Y 495.734,Z 225.229,A -85,B 0,C 180,E1 -6044.786,E2 -6044.786} C_VEL
LIN {X 0,Y 495.726,Z 225.231,A -85,B 0,C 180,E1 -6048.175,E2 -6048.175} C_VEL
LIN {X 0,Y 495.705,Z 225.232,A -85,B 0,C 180,E1 -6050.761,E2 -6050.761} C_VEL
LIN {X 0,Y 495.691,Z 225.237,A -85,B 0,C 180,E1 -6053.391,E2 -6053.391} C_VEL
LIN {X 0,Y 495.739,Z 225.234,A -85,B 0,C 180,E1 -6056.072,E2 -6056.072} C_VEL
LIN {X 0,Y 495.718,Z 225.23,A -85,B 0,C 180,E1 -6058.819,E2 -6058.819} C_VEL
LIN {X 0,Y 495.705,Z 225.236,A -85,B 0,C 180,E1 -6061.732,E2 -6061.732} C_VEL
LIN {X 0,Y 495.72,Z 225.232,A -85,B 0,C 180,E1 -6064.701,E2 -6064.701} C_VEL
LIN {X 0,Y 495.678,Z 225.236,A -85,B 0,C 180,E1 -6067.567,E2 -6067.567} C_VEL
LIN {X 0,Y 495.731,Z 225.233,A -85,B 0,C 180,E1 -6070.704,E2 -6070.704} C_VEL
LIN {X 0,Y 495.688,Z 225.234,A -85,B 0,C 180,E1 -6073.702,E2 -6073.702} C_VEL
LIN {X 0,Y 495.692,Z 225.239,A -85,B 0,C 180,E1 -6076.311,E2 -6076.311} C_VEL
LIN {X 0,Y 495.743,Z 225.229,A -85,B 0,C 180,E1 -6079.308,E2 -6079.308} C_VEL
LIN {X 0,Y 495.695,Z 225.237,A -85,B 0,C 180,E1 -6082.445,E2 -6082.445} C_VEL
LIN {X 0,Y 495.745,Z 225.229,A -85,B 0,C 180,E1 -6085.463,E2 -6085.463} C_VEL
LIN {X 0,Y 495.726,Z 225.231,A -85,B 0,C 180,E1 -6088.37,E2 -6088.37} C_VEL
LIN {X 0,Y 495.762,Z 225.228,A -85,B 0,C 180,E1 -6091.514,E2 -6091.514} C_VEL
LIN {X 0,Y 495.768,Z 225.225,A -85,B 0,C 180,E1 -6093.939,E2 -6093.939} C_VEL
LIN {X 0,Y 495.742,Z 225.235,A -85,B 0,C 180,E1 -6097.146,E2 -6097.146} C_VEL
LIN {X 0,Y 495.755,Z 225.226,A -85,B 0,C 180,E1 -6100.116,E2 -6100.116} C_VEL
LIN {X 0,Y 495.751,Z 225.227,A -85,B 0,C 180,E1 -6102.687,E2 -6102.687} C_VEL
LIN {X 0,Y 495.78,Z 225.227,A -85,B 0,C 180,E1 -6105.223,E2 -6105.223} C_VEL
LIN {X 0,Y 495.845,Z 225.215,A -85,B 0,C 180,E1 -6108.561,E2 -6108.561} C_VEL
LIN {X 0,Y 495.834,Z 225.225,A -85,B 0,C 180,E1 -6111.857,E2 -6111.857} C_VEL
LIN {X 0,Y 495.864,Z 225.215,A -85,B 0,C 180,E1 -6114.312,E2 -6114.312} C_VEL
LIN {X 0,Y 495.987,Z 225.2,A -85,B 0,C 180,E1 -6117.569,E2 -6117.569} C_VEL
LIN {X 0,Y 495.927,Z 225.205,A -85,B 0,C 180,E1 -6120.817,E2 -6120.817} C_VEL
LIN {X 0,Y 495.982,Z 225.202,A -85,B 0,C 180,E1 -6122.442,E2 -6122.442} C_VEL
LIN {X 0,Y 495.868,Z 225.213,A -85,B 0,C 180,E1 -6125.699,E2 -6125.699} C_VEL
LIN {X 0,Y 495.822,Z 225.224,A -85,B 0,C 180,E1 -6128.154,E2 -6128.154} C_VEL
LIN {X 0,Y 495.861,Z 225.212,A -85,B 0,C 180,E1 -6131.45,E2 -6131.45} C_VEL
LIN {X 0,Y 495.792,Z 225.227,A -85,B 0,C 180,E1 -6134.787,E2 -6134.787} C_VEL
LIN {X 0,Y 495.77,Z 225.225,A -85,B 0,C 180,E1 -6137.324,E2 -6137.324} C_VEL
LIN {X 0,Y 495.776,Z 225.223,A -85,B 0,C 180,E1 -6139.894,E2 -6139.894} C_VEL
LIN {X 0,Y 495.775,Z 225.233,A -85,B 0,C 180,E1 -6142.863,E2 -6142.863} C_VEL
LIN {X 0,Y 495.734,Z 225.228,A -85,B 0,C 180,E1 -6146.075,E2 -6146.075} C_VEL
LIN {X 0,Y 495.746,Z 225.233,A -85,B 0,C 180,E1 -6148.82,E2 -6148.82} C_VEL
LIN {X 0,Y 495.768,Z 225.226,A -85,B 0,C 180,E1 -6151.726,E2 -6151.726} C_VEL
LIN {X 0,Y 495.775,Z 225.225,A -85,B 0,C 180,E1 -6154.694,E2 -6154.694} C_VEL
LIN {X 0,Y 495.738,Z 225.234,A -85,B 0,C 180,E1 -6157.565,E2 -6157.565} C_VEL
LIN {X 0,Y 495.763,Z 225.226,A -85,B 0,C 180,E1 -6160.046,E2 -6160.046} C_VEL
LIN {X 0,Y 495.709,Z 225.233,A -85,B 0,C 180,E1 -6162.888,E2 -6162.888} C_VEL
LIN {X 0,Y 495.732,Z 225.232,A -85,B 0,C 180,E1 -6165.998,E2 -6165.998} C_VEL
LIN {X 0,Y 495.745,Z 225.23,A -85,B 0,C 180,E1 -6169.297,E2 -6169.297} C_VEL
LIN {X 0,Y 495.742,Z 225.231,A -85,B 0,C 180,E1 -6171.407,E2 -6171.407} C_VEL
LIN {X 0,Y 495.759,Z 225.227,A -85,B 0,C 180,E1 -6174.462,E2 -6174.462} C_VEL
LIN {X 0,Y 495.769,Z 225.225,A -85,B 0,C 180,E1 -6177.405,E2 -6177.405} C_VEL
LIN {X 0,Y 495.779,Z 225.232,A -85,B 0,C 180,E1 -6180.253,E2 -6180.253} C_VEL
LIN {X 0,Y 495.791,Z 225.226,A -85,B 0,C 180,E1 -6183.262,E2 -6183.262} C_VEL
LIN {X 0,Y 495.813,Z 225.357,A -85,B 0,C 180,E1 -6185.838,E2 -6185.838} C_VEL
LIN {X 0,Y 497.386,Z 234.269,A -85,B 0,C 180,E1 -6187.572,E2 -6187.572} C_VEL
LIN {X 0,Y 497.075,Z 245.112,A -85,B 0,C 180,E1 -6189.516,E2 -6189.516} C_VEL
LIN {X 0,Y 496.53,Z 261.99,A -85,B 0,C 180,E1 -6192.495,E2 -6192.495} C_VEL
LIN {X 0,Y 496.315,Z 270.539,A -85,B 0,C 180,E1 -6193.954,E2 -6193.954} C_VEL
LIN {X 0,Y 497.989,Z 280.761,A -85,B 0,C 180,E1 -6194.192,E2 -6194.192} C_VEL
LIN {X 0,Y 498.532,Z 287.038,A -85,B 0,C 180,E1 -6194.304,E2 -6194.304} C_VEL
LIN {X 0,Y 497.924,Z 378.603,A -85,B 0,C 180,E1 -6195.672,E2 -6195.672} C_VEL
LIN {X 0,Y 497.62,Z 392.465,A -85,B 0,C 180,E1 -6196.055,E2 -6196.055} C_VEL
LIN {X 0,Y 497.285,Z 404.906,A -85,B 0,C 180,E1 -6196.566,E2 -6196.566} C_VEL
LIN {X 0,Y 496.929,Z 416.917,A -85,B 0,C 180,E1 -6197.239,E2 -6197.239} C_VEL
LIN {X 0,Y 496.594,Z 428.243,A -85,B 0,C 180,E1 -6198.053,E2 -6198.053} C_VEL
LIN {X 0,Y 496.192,Z 438.553,A -85,B 0,C 180,E1 -6198.975,E2 -6198.975} C_VEL
LIN {X 0,Y 495.839,Z 447.804,A -85,B 0,C 180,E1 -6200,E2 -6200} C_VEL
LIN {X 0,Y 495.549,Z 456.793,A -85,B 0,C 180,E1 -6201.229,E2 -6201.229} C_VEL
LIN {X 0,Y 495.315,Z 464.028,A -85,B 0,C 180,E1 -6202.457,E2 -6202.457} C_VEL
LIN {X 0,Y 495.147,Z 470.07,A -85,B 0,C 180,E1 -6203.75,E2 -6203.75} C_VEL
LIN {X 0,Y 495.04,Z 474.97,A -85,B 0,C 180,E1 -6205.112,E2 -6205.112} C_VEL
LIN {X 0,Y 495.035,Z 477.273,A -85,B 0,C 180,E1 -6205.928,E2 -6205.928} C_VEL
LIN {X 0,Y 495.045,Z 479.142,A -85,B 0,C 180,E1 -6206.743,E2 -6206.743} C_VEL
LIN {X 0,Y 494.964,Z 481.541,A -85,B 0,C 180,E1 -6208.371,E2 -6208.371} C_VEL
LIN {X 0,Y 494.901,Z 482.365,A -85,B 0,C 180,E1 -6209.999,E2 -6209.999} C_VEL
LIN {X 0,Y 494.963,Z 481.537,A -85,B 0,C 180,E1 -6211.626,E2 -6211.626} C_VEL
LIN {X 0,Y 495.045,Z 479.134,A -85,B 0,C 180,E1 -6213.254,E2 -6213.254} C_VEL
LIN {X 0,Y 495.01,Z 476.185,A -85,B 0,C 180,E1 -6214.477,E2 -6214.477} C_VEL
LIN {X 0,Y 495.145,Z 472.193,A -85,B 0,C 180,E1 -6215.701,E2 -6215.701} C_VEL
LIN {X 0,Y 495.245,Z 466.046,A -85,B 0,C 180,E1 -6217.131,E2 -6217.131} C_VEL
LIN {X 0,Y 495.439,Z 459.334,A -85,B 0,C 180,E1 -6218.359,E2 -6218.359} C_VEL
LIN {X 0,Y 495.72,Z 451.004,A -85,B 0,C 180,E1 -6219.588,E2 -6219.588} C_VEL
LIN {X 0,Y 495.98,Z 442.438,A -85,B 0,C 180,E1 -6220.613,E2 -6220.613} C_VEL
LIN {X 0,Y 496.434,Z 431.863,A -85,B 0,C 180,E1 -6221.637,E2 -6221.637} C_VEL
LIN {X 0,Y 496.773,Z 420.408,A -85,B 0,C 180,E1 -6222.528,E2 -6222.528} C_VEL
LIN {X 0,Y 497.147,Z 409.853,A -85,B 0,C 180,E1 -6223.175,E2 -6223.175} C_VEL
LIN {X 0,Y 497.479,Z 397.895,A -85,B 0,C 180,E1 -6223.738,E2 -6223.738} C_VEL
LIN {X 0,Y 497.818,Z 384.085,A -85,B 0,C 180,E1 -6224.198,E2 -6224.198} C_VEL
LIN {X 0,Y 497.996,Z 371.403,A -85,B 0,C 180,E1 -6224.453,E2 -6224.453} C_VEL
LIN {X 0,Y 498.519,Z 284.36,A -85,B 0,C 180,E1 -6225.741,E2 -6225.741} C_VEL
LIN {X 0,Y 496.266,Z 270.265,A -85,B 0,C 180,E1 -6226.053,E2 -6226.053} C_VEL
LIN {X 0,Y 496.737,Z 253.019,A -85,B 0,C 180,E1 -6228.989,E2 -6228.989} C_VEL
LIN {X 0,Y 497.269,Z 235.764,A -85,B 0,C 180,E1 -6231.993,E2 -6231.993} C_VEL
LIN {X 0,Y 496.95,Z 231.521,A -85,B 0,C 180,E1 -6232.759,E2 -6232.759} C_VEL
LIN {X 0,Y 495.804,Z 225.321,A -85,B 0,C 180,E1 -6233.965,E2 -6233.965} C_VEL
LIN {X 0,Y 495.79,Z 225.226,A -85,B 0,C 180,E1 -6236.974,E2 -6236.974} C_VEL
LIN {X 0,Y 495.771,Z 225.233,A -85,B 0,C 180,E1 -6239.744,E2 -6239.744} C_VEL
LIN {X 0,Y 495.772,Z 225.227,A -85,B 0,C 180,E1 -6242.592,E2 -6242.592} C_VEL
LIN {X 0,Y 495.749,Z 225.232,A -85,B 0,C 180,E1 -6245.535,E2 -6245.535} C_VEL
LIN {X 0,Y 495.76,Z 225.227,A -85,B 0,C 180,E1 -6248.764,E2 -6248.764} C_VEL
LIN {X 0,Y 495.728,Z 225.234,A -85,B 0,C 180,E1 -6251.781,E2 -6251.781} C_VEL
LIN {X 0,Y 495.739,Z 225.228,A -85,B 0,C 180,E1 -6255.138,E2 -6255.138} C_VEL
LIN {X 0,Y 495.725,Z 225.237,A -85,B 0,C 180,E1 -6258.212,E2 -6258.212} C_VEL
LIN {X 0,Y 495.74,Z 225.228,A -85,B 0,C 180,E1 -6261.232,E2 -6261.232} C_VEL
LIN {X 0,Y 495.728,Z 225.237,A -85,B 0,C 180,E1 -6264.457,E2 -6264.457} C_VEL
LIN {X 0,Y 495.749,Z 225.227,A -85,B 0,C 180,E1 -6267.401,E2 -6267.401} C_VEL
LIN {X 0,Y 495.754,Z 225.231,A -85,B 0,C 180,E1 -6270.249,E2 -6270.249} C_VEL
LIN {X 0,Y 495.735,Z 225.227,A -85,B 0,C 180,E1 -6273.267,E2 -6273.267} C_VEL
LIN {X 0,Y 495.703,Z 225.233,A -85,B 0,C 180,E1 -6275.718,E2 -6275.718} C_VEL
LIN {X 0,Y 495.722,Z 225.233,A -85,B 0,C 180,E1 -6278.366,E2 -6278.366} C_VEL
LIN {X 0,Y 495.743,Z 225.233,A -85,B 0,C 180,E1 -6280.966,E2 -6280.966} C_VEL
LIN {X 0,Y 495.778,Z 225.227,A -85,B 0,C 180,E1 -6284.56,E2 -6284.56} C_VEL
LIN {X 0,Y 495.817,Z 225.216,A -85,B 0,C 180,E1 -6287.961,E2 -6287.961} C_VEL
LIN {X 0,Y 495.784,Z 225.229,A -85,B 0,C 180,E1 -6291.024,E2 -6291.024} C_VEL
LIN {X 0,Y 495.828,Z 225.22,A -85,B 0,C 180,E1 -6293.484,E2 -6293.484} C_VEL
LIN {X 0,Y 495.689,Z 225.236,A -85,B 0,C 180,E1 -6295.93,E2 -6295.93} C_VEL
LIN {X 0,Y 495.963,Z 225.205,A -85,B 0,C 180,E1 -6297.558,E2 -6297.558} C_VEL
LIN {X 0,Y 495.974,Z 225.199,A -85,B 0,C 180,E1 -6299.995,E2 -6299.995} C_VEL
LIN {X 0,Y 495.969,Z 225.199,A -85,B 0,C 180,E1 -6302.431,E2 -6302.431} C_VEL
LIN {X 0,Y 495.862,Z 225.219,A -85,B 0,C 180,E1 -6305.688,E2 -6305.688} C_VEL
LIN {X 0,Y 495.817,Z 225.222,A -85,B 0,C 180,E1 -6308.964,E2 -6308.964} C_VEL
LIN {X 0,Y 495.825,Z 225.22,A -85,B 0,C 180,E1 -6312.269,E2 -6312.269} C_VEL
LIN {X 0,Y 495.776,Z 225.233,A -85,B 0,C 180,E1 -6315.618,E2 -6315.618} C_VEL
LIN {X 0,Y 495.772,Z 225.229,A -85,B 0,C 180,E1 -6318.242,E2 -6318.242} C_VEL
LIN {X 0,Y 495.741,Z 225.231,A -85,B 0,C 180,E1 -6320.751,E2 -6320.751} C_VEL
LIN {X 0,Y 495.744,Z 225.235,A -85,B 0,C 180,E1 -6323.38,E2 -6323.38} C_VEL
LIN {X 0,Y 495.84,Z 225.274,A -85,B 0,C 180,E1 -6324.355,E2 -6324.355} C_VEL
LIN {X 0,Y 496.686,Z 230.339,A -85,B 0,C 180,E1 -6325.335,E2 -6325.335} C_VEL
LIN {X 0,Y 496.362,Z 248.1,A -85,B 0,C 180,E1 -6328.421,E2 -6328.421} C_VEL
LIN {X 0,Y 496.273,Z 257.219,A -85,B 0,C 180,E1 -6329.987,E2 -6329.987} C_VEL
LIN {X 0,Y 497.83,Z 266.185,A -85,B 0,C 180,E1 -6330.204,E2 -6330.204} C_VEL
LIN {X 0,Y 498.566,Z 272.22,A -85,B 0,C 180,E1 -6330.321,E2 -6330.321} C_VEL
LIN {X 0,Y 497.916,Z 365.577,A -85,B 0,C 180,E1 -6331.725,E2 -6331.725} C_VEL
LIN {X 0,Y 497.673,Z 379.193,A -85,B 0,C 180,E1 -6332.106,E2 -6332.106} C_VEL
LIN {X 0,Y 497.369,Z 392.16,A -85,B 0,C 180,E1 -6332.648,E2 -6332.648} C_VEL
LIN {X 0,Y 497.047,Z 403.56,A -85,B 0,C 180,E1 -6333.293,E2 -6333.293} C_VEL
LIN {X 0,Y 496.611,Z 414.781,A -85,B 0,C 180,E1 -6334.1,E2 -6334.1} C_VEL
LIN {X 0,Y 496.248,Z 424.848,A -85,B 0,C 180,E1 -6335.002,E2 -6335.002} C_VEL
LIN {X 0,Y 495.937,Z 433.523,A -85,B 0,C 180,E1 -6335.954,E2 -6335.954} C_VEL
LIN {X 0,Y 495.593,Z 442.721,A -85,B 0,C 180,E1 -6337.2,E2 -6337.2} C_VEL
LIN {X 0,Y 495.395,Z 449.609,A -85,B 0,C 180,E1 -6338.355,E2 -6338.355} C_VEL
LIN {X 0,Y 495.183,Z 455.97,A -85,B 0,C 180,E1 -6339.683,E2 -6339.683} C_VEL
LIN {X 0,Y 495.086,Z 460.024,A -85,B 0,C 180,E1 -6340.76,E2 -6340.76} C_VEL
LIN {X 0,Y 494.383,Z 462.066,A -85,B 0,C 180,E1 -6341.399,E2 -6341.399} C_VEL
LIN {X 0,Y 491.441,Z 464.827,A -85,B 0,C 180,E1 -6342.451,E2 -6342.451} C_VEL
LIN {X 0,Y 488.966,Z 466.541,A -85,B 0,C 180,E1 -6343.314,E2 -6343.314} C_VEL
LIN {X 0,Y 487.836,Z 467.656,A -85,B 0,C 180,E1 -6344.104,E2 -6344.104} C_VEL
LIN {X 0,Y 487.812,Z 467.71,A -85,B 0,C 180,E1 -6344.219,E2 -6344.219} C_VEL
LIN {X 0,Y 487.831,Z 468.47,A -85,B 0,C 180,E1 -6345.099,E2 -6345.099} C_VEL
LIN {X 0,Y 487.766,Z 468.72,A -85,B 0,C 180,E1 -6346.245,E2 -6346.245} C_VEL
LIN {X 0,Y 487.818,Z 468.223,A -85,B 0,C 180,E1 -6347.383,E2 -6347.383} C_VEL
LIN {X 0,Y 487.862,Z 466.955,A -85,B 0,C 180,E1 -6348.499,E2 -6348.499} C_VEL
LIN {X 0,Y 487.873,Z 464.641,A -85,B 0,C 180,E1 -6349.759,E2 -6349.759} C_VEL
LIN {X 0,Y 487.955,Z 461.246,A -85,B 0,C 180,E1 -6351.042,E2 -6351.042} C_VEL
LIN {X 0,Y 488.108,Z 456.607,A -85,B 0,C 180,E1 -6352.351,E2 -6352.351} C_VEL
LIN {X 0,Y 488.285,Z 450.456,A -85,B 0,C 180,E1 -6353.694,E2 -6353.694} C_VEL
LIN {X 0,Y 488.576,Z 442.436,A -85,B 0,C 180,E1 -6355.062,E2 -6355.062} C_VEL
LIN {X 0,Y 488.882,Z 434.072,A -85,B 0,C 180,E1 -6356.211,E2 -6356.211} C_VEL
LIN {X 0,Y 489.255,Z 424.401,A -85,B 0,C 180,E1 -6357.287,E2 -6357.287} C_VEL
LIN {X 0,Y 489.698,Z 413.101,A -85,B 0,C 180,E1 -6358.291,E2 -6358.291} C_VEL
LIN {X 0,Y 490.078,Z 402.65,A -85,B 0,C 180,E1 -6359.035,E2 -6359.035} C_VEL
LIN {X 0,Y 490.488,Z 390.555,A -85,B 0,C 180,E1 -6359.705,E2 -6359.705} C_VEL
LIN {X 0,Y 490.778,Z 377.255,A -85,B 0,C 180,E1 -6360.243,E2 -6360.243} C_VEL
LIN {X 0,Y 491.067,Z 364.639,A -85,B 0,C 180,E1 -6360.582,E2 -6360.582} C_VEL
LIN {X 0,Y 491.65,Z 271.106,A -85,B 0,C 180,E1 -6362.001,E2 -6362.001} C_VEL
LIN {X 0,Y 489.382,Z 258.094,A -85,B 0,C 180,E1 -6362.296,E2 -6362.296} C_VEL
LIN {X 0,Y 489.409,Z 255.927,A -85,B 0,C 180,E1 -6362.646,E2 -6362.646} C_VEL
LIN {X 0,Y 489.992,Z 239.458,A -85,B 0,C 180,E1 -6365.874,E2 -6365.874} C_VEL
LIN {X 0,Y 489.983,Z 232.737,A -85,B 0,C 180,E1 -6367.217,E2 -6367.217} C_VEL
LIN {X 0,Y 488.696,Z 226.183,A -85,B 0,C 180,E1 -6368.654,E2 -6368.654} C_VEL
LIN {X 0,Y 488.681,Z 226.112,A -85,B 0,C 180,E1 -6371.626,E2 -6371.626} C_VEL
LIN {X 0,Y 488.711,Z 226.106,A -85,B 0,C 180,E1 -6375,E2 -6375} C_VEL
LIN {X 0,Y 488.758,Z 226.103,A -85,B 0,C 180,E1 -6378.388,E2 -6378.388} C_VEL
LIN {X 0,Y 488.748,Z 226.099,A -85,B 0,C 180,E1 -6381.734,E2 -6381.734} C_VEL
LIN {X 0,Y 488.798,Z 226.094,A -85,B 0,C 180,E1 -6384.225,E2 -6384.225} C_VEL
LIN {X 0,Y 488.891,Z 226.082,A -85,B 0,C 180,E1 -6387.53,E2 -6387.53} C_VEL
LIN {X 0,Y 488.887,Z 226.081,A -85,B 0,C 180,E1 -6390.001,E2 -6390.001} C_VEL
LIN {X 0,Y 488.891,Z 226.082,A -85,B 0,C 180,E1 -6392.473,E2 -6392.473} C_VEL
LIN {X 0,Y 488.799,Z 226.094,A -85,B 0,C 180,E1 -6395.778,E2 -6395.778} C_VEL
LIN {X 0,Y 488.751,Z 226.098,A -85,B 0,C 180,E1 -6398.269,E2 -6398.269} C_VEL
LIN {X 0,Y 488.763,Z 226.103,A -85,B 0,C 180,E1 -6401.615,E2 -6401.615} C_VEL
LIN {X 0,Y 488.701,Z 226.107,A -85,B 0,C 180,E1 -6405.004,E2 -6405.004} C_VEL
LIN {X 0,Y 488.685,Z 226.107,A -85,B 0,C 180,E1 -6408.446,E2 -6408.446} C_VEL
LIN {X 0,Y 488.64,Z 226.113,A -85,B 0,C 180,E1 -6411.075,E2 -6411.075} C_VEL
LIN {X 0,Y 488.634,Z 226.121,A -85,B 0,C 180,E1 -6413.75,E2 -6413.75} C_VEL
LIN {X 0,Y 488.735,Z 226.1,A -85,B 0,C 180,E1 -6416.95,E2 -6416.95} C_VEL
LIN {X 0,Y 488.663,Z 226.114,A -85,B 0,C 180,E1 -6420.371,E2 -6420.371} C_VEL
LIN {X 0,Y 488.679,Z 226.108,A -85,B 0,C 180,E1 -6423.49,E2 -6423.49} C_VEL
LIN {X 0,Y 488.634,Z 226.12,A -85,B 0,C 180,E1 -6426.361,E2 -6426.361} C_VEL
LIN {X 0,Y 488.691,Z 226.106,A -85,B 0,C 180,E1 -6429.256,E2 -6429.256} C_VEL
LIN {X 0,Y 488.686,Z 226.115,A -85,B 0,C 180,E1 -6432.527,E2 -6432.527} C_VEL
LIN {X 0,Y 488.667,Z 226.11,A -85,B 0,C 180,E1 -6435.205,E2 -6435.205} C_VEL
LIN {X 0,Y 488.692,Z 226.106,A -85,B 0,C 180,E1 -6437.485,E2 -6437.485} C_VEL
LIN {X 0,Y 488.71,Z 226.113,A -85,B 0,C 180,E1 -6440.757,E2 -6440.757} C_VEL
LIN {X 0,Y 488.65,Z 226.111,A -85,B 0,C 180,E1 -6443.875,E2 -6443.875} C_VEL
LIN {X 0,Y 488.706,Z 226.113,A -85,B 0,C 180,E1 -6446.884,E2 -6446.884} C_VEL
LIN {X 0,Y 488.697,Z 226.106,A -85,B 0,C 180,E1 -6449.787,E2 -6449.787} C_VEL
LIN {X 0,Y 488.769,Z 226.104,A -85,B 0,C 180,E1 -6453.063,E2 -6453.063} C_VEL
LIN {X 0,Y 488.669,Z 226.108,A -85,B 0,C 180,E1 -6456.261,E2 -6456.261} C_VEL
LIN {X 0,Y 488.731,Z 226.107,A -85,B 0,C 180,E1 -6459.182,E2 -6459.182} C_VEL
LIN {X 0,Y 488.737,Z 226.106,A -85,B 0,C 180,E1 -6461.638,E2 -6461.638} C_VEL
LIN {X 0,Y 488.752,Z 226.1,A -85,B 0,C 180,E1 -6465.006,E2 -6465.006} C_VEL
LIN {X 0,Y 488.8,Z 226.093,A -85,B 0,C 180,E1 -6468.394,E2 -6468.394} C_VEL
LIN {X 0,Y 488.783,Z 226.103,A -85,B 0,C 180,E1 -6471.739,E2 -6471.739} C_VEL
LIN {X 0,Y 488.824,Z 226.093,A -85,B 0,C 180,E1 -6474.23,E2 -6474.23} C_VEL
LIN {X 0,Y 488.954,Z 226.076,A -85,B 0,C 180,E1 -6477.534,E2 -6477.534} C_VEL
LIN {X 0,Y 488.88,Z 226.083,A -85,B 0,C 180,E1 -6480.829,E2 -6480.829} C_VEL
LIN {X 0,Y 488.948,Z 226.078,A -85,B 0,C 180,E1 -6482.477,E2 -6482.477} C_VEL
LIN {X 0,Y 488.827,Z 226.091,A -85,B 0,C 180,E1 -6485.781,E2 -6485.781} C_VEL
LIN {X 0,Y 488.769,Z 226.104,A -85,B 0,C 180,E1 -6488.272,E2 -6488.272} C_VEL
LIN {X 0,Y 488.816,Z 226.09,A -85,B 0,C 180,E1 -6491.617,E2 -6491.617} C_VEL
LIN {X 0,Y 488.769,Z 226.099,A -85,B 0,C 180,E1 -6495.005,E2 -6495.005} C_VEL
LIN {X 0,Y 488.761,Z 226.103,A -85,B 0,C 180,E1 -6498.446,E2 -6498.446} C_VEL
LIN {X 0,Y 488.723,Z 226.107,A -85,B 0,C 180,E1 -6501.074,E2 -6501.074} C_VEL
LIN {X 0,Y 488.685,Z 226.107,A -85,B 0,C 180,E1 -6503.75,E2 -6503.75} C_VEL
LIN {X 0,Y 488.716,Z 226.111,A -85,B 0,C 180,E1 -6506.924,E2 -6506.924} C_VEL
LIN {X 0,Y 488.735,Z 226.1,A -85,B 0,C 180,E1 -6510.222,E2 -6510.222} C_VEL
LIN {X 0,Y 488.729,Z 226.106,A -85,B 0,C 180,E1 -6513.482,E2 -6513.482} C_VEL
LIN {X 0,Y 488.688,Z 226.106,A -85,B 0,C 180,E1 -6516.354,E2 -6516.354} C_VEL
LIN {X 0,Y 488.713,Z 226.11,A -85,B 0,C 180,E1 -6519.257,E2 -6519.257} C_VEL
LIN {X 0,Y 488.686,Z 226.114,A -85,B 0,C 180,E1 -6521.596,E2 -6521.596} C_VEL
LIN {X 0,Y 488.714,Z 226.103,A -85,B 0,C 180,E1 -6524.805,E2 -6524.805} C_VEL
LIN {X 0,Y 488.667,Z 226.115,A -85,B 0,C 180,E1 -6527.471,E2 -6527.471} C_VEL
LIN {X 0,Y 488.723,Z 226.11,A -85,B 0,C 180,E1 -6529.674,E2 -6529.674} C_VEL
LIN {X 0,Y 488.679,Z 226.107,A -85,B 0,C 180,E1 -6532.84,E2 -6532.84} C_VEL
LIN {X 0,Y 488.735,Z 226.109,A -85,B 0,C 180,E1 -6535.886,E2 -6535.886} C_VEL
LIN {X 0,Y 488.707,Z 226.104,A -85,B 0,C 180,E1 -6538.82,E2 -6538.82} C_VEL
LIN {X 0,Y 488.73,Z 226.106,A -85,B 0,C 180,E1 -6541.669,E2 -6541.669} C_VEL
LIN {X 0,Y 488.717,Z 226.11,A -85,B 0,C 180,E1 -6544.441,E2 -6544.441} C_VEL
LIN {X 0,Y 488.759,Z 226.198,A -85,B 0,C 180,E1 -6545.636,E2 -6545.636} C_VEL
LIN {X 0,Y 490.411,Z 235.373,A -85,B 0,C 180,E1 -6547.458,E2 -6547.458} C_VEL
LIN {X 0,Y 490.171,Z 245.023,A -85,B 0,C 180,E1 -6549.214,E2 -6549.214} C_VEL
LIN {X 0,Y 489.534,Z 263.09,A -85,B 0,C 180,E1 -6552.452,E2 -6552.452} C_VEL
LIN {X 0,Y 489.325,Z 270.344,A -85,B 0,C 180,E1 -6553.712,E2 -6553.712} C_VEL
LIN {X 0,Y 489.963,Z 274.69,A -85,B 0,C 180,E1 -6553.841,E2 -6553.841} C_VEL
LIN {X 0,Y 491.691,Z 286.597,A -85,B 0,C 180,E1 -6554.08,E2 -6554.08} C_VEL
LIN {X 0,Y 491.054,Z 378.181,A -85,B 0,C 180,E1 -6555.467,E2 -6555.467} C_VEL
LIN {X 0,Y 490.747,Z 391.384,A -85,B 0,C 180,E1 -6555.829,E2 -6555.829} C_VEL
LIN {X 0,Y 490.364,Z 404.648,A -85,B 0,C 180,E1 -6556.373,E2 -6556.373} C_VEL
LIN {X 0,Y 489.992,Z 416.597,A -85,B 0,C 180,E1 -6557.048,E2 -6557.048} C_VEL
LIN {X 0,Y 489.622,Z 428.049,A -85,B 0,C 180,E1 -6557.881,E2 -6557.881} C_VEL
LIN {X 0,Y 489.208,Z 438.38,A -85,B 0,C 180,E1 -6558.816,E2 -6558.816} C_VEL
LIN {X 0,Y 488.824,Z 447.649,A -85,B 0,C 180,E1 -6559.855,E2 -6559.855} C_VEL
LIN {X 0,Y 488.478,Z 456.651,A -85,B 0,C 180,E1 -6561.101,E2 -6561.101} C_VEL
LIN {X 0,Y 488.247,Z 463.9,A -85,B 0,C 180,E1 -6562.347,E2 -6562.347} C_VEL
LIN {X 0,Y 488.05,Z 470.419,A -85,B 0,C 180,E1 -6563.778,E2 -6563.778} C_VEL
LIN {X 0,Y 487.971,Z 474.862,A -85,B 0,C 180,E1 -6565.041,E2 -6565.041} C_VEL
LIN {X 0,Y 487.931,Z 477.167,A -85,B 0,C 180,E1 -6565.869,E2 -6565.869} C_VEL
LIN {X 0,Y 487.968,Z 479.04,A -85,B 0,C 180,E1 -6566.696,E2 -6566.696} C_VEL
LIN {X 0,Y 487.892,Z 481.441,A -85,B 0,C 180,E1 -6568.348,E2 -6568.348} C_VEL
LIN {X 0,Y 487.822,Z 482.267,A -85,B 0,C 180,E1 -6569.999,E2 -6569.999} C_VEL
LIN {X 0,Y 487.892,Z 481.438,A -85,B 0,C 180,E1 -6571.649,E2 -6571.649} C_VEL
LIN {X 0,Y 487.968,Z 479.033,A -85,B 0,C 180,E1 -6573.301,E2 -6573.301} C_VEL
LIN {X 0,Y 487.923,Z 476.081,A -85,B 0,C 180,E1 -6574.542,E2 -6574.542} C_VEL
LIN {X 0,Y 488.062,Z 472.087,A -85,B 0,C 180,E1 -6575.784,E2 -6575.784} C_VEL
LIN {X 0,Y 488.182,Z 465.937,A -85,B 0,C 180,E1 -6577.235,E2 -6577.235} C_VEL
LIN {X 0,Y 488.387,Z 459.219,A -85,B 0,C 180,E1 -6578.481,E2 -6578.481} C_VEL
LIN {X 0,Y 488.706,Z 450.881,A -85,B 0,C 180,E1 -6579.727,E2 -6579.727} C_VEL
LIN {X 0,Y 488.987,Z 442.306,A -85,B 0,C 180,E1 -6580.767,E2 -6580.767} C_VEL
LIN {X 0,Y 489.468,Z 431.722,A -85,B 0,C 180,E1 -6581.805,E2 -6581.805} C_VEL
LIN {X 0,Y 489.786,Z 421.216,A -85,B 0,C 180,E1 -6582.64,E2 -6582.64} C_VEL
LIN {X 0,Y 490.212,Z 409.682,A -85,B 0,C 180,E1 -6583.365,E2 -6583.365} C_VEL
LIN {X 0,Y 490.563,Z 397.702,A -85,B 0,C 180,E1 -6583.936,E2 -6583.936} C_VEL
LIN {X 0,Y 490.929,Z 384.776,A -85,B 0,C 180,E1 -6584.375,E2 -6584.375} C_VEL
LIN {X 0,Y 491.129,Z 371.093,A -85,B 0,C 180,E1 -6584.66,E2 -6584.66} C_VEL
LIN {X 0,Y 491.613,Z 284.463,A -85,B 0,C 180,E1 -6585.967,E2 -6585.967} C_VEL
LIN {X 0,Y 489.271,Z 270.158,A -85,B 0,C 180,E1 -6586.293,E2 -6586.293} C_VEL
LIN {X 0,Y 489.763,Z 253.913,A -85,B 0,C 180,E1 -6589.092,E2 -6589.092} C_VEL
LIN {X 0,Y 490.335,Z 236.881,A -85,B 0,C 180,E1 -6592.099,E2 -6592.099} C_VEL
LIN {X 0,Y 490.053,Z 233.158,A -85,B 0,C 180,E1 -6592.779,E2 -6592.779} C_VEL
LIN {X 0,Y 488.754,Z 226.244,A -85,B 0,C 180,E1 -6594.135,E2 -6594.135} C_VEL
LIN {X 0,Y 488.737,Z 226.108,A -85,B 0,C 180,E1 -6597.395,E2 -6597.395} C_VEL
LIN {X 0,Y 488.713,Z 226.106,A -85,B 0,C 180,E1 -6600.36,E2 -6600.36} C_VEL
LIN {X 0,Y 488.739,Z 226.106,A -85,B 0,C 180,E1 -6603.481,E2 -6603.481} C_VEL
LIN {X 0,Y 488.677,Z 226.114,A -85,B 0,C 180,E1 -6606.35,E2 -6606.35} C_VEL
LIN {X 0,Y 488.696,Z 226.107,A -85,B 0,C 180,E1 -6609.252,E2 -6609.252} C_VEL
LIN {X 0,Y 488.669,Z 226.112,A -85,B 0,C 180,E1 -6612.525,E2 -6612.525} C_VEL
LIN {X 0,Y 488.703,Z 226.105,A -85,B 0,C 180,E1 -6615.194,E2 -6615.194} C_VEL
LIN {X 0,Y 488.663,Z 226.115,A -85,B 0,C 180,E1 -6618.576,E2 -6618.576} C_VEL
LIN {X 0,Y 488.688,Z 226.108,A -85,B 0,C 180,E1 -6620.946,E2 -6620.946} C_VEL
LIN {X 0,Y 488.645,Z 226.113,A -85,B 0,C 180,E1 -6623.861,E2 -6623.861} C_VEL
LIN {X 0,Y 488.709,Z 226.109,A -85,B 0,C 180,E1 -6626.517,E2 -6626.517} C_VEL
LIN {X 0,Y 488.713,Z 226.104,A -85,B 0,C 180,E1 -6629.776,E2 -6629.776} C_VEL
LIN {X 0,Y 488.693,Z 226.106,A -85,B 0,C 180,E1 -6633.075,E2 -6633.075} C_VEL
LIN {X 0,Y 488.69,Z 226.108,A -85,B 0,C 180,E1 -6635.347,E2 -6635.347} C_VEL
LIN {X 0,Y 488.678,Z 226.107,A -85,B 0,C 180,E1 -6638.038,E2 -6638.038} C_VEL
LIN {X 0,Y 488.701,Z 226.111,A -85,B 0,C 180,E1 -6640.681,E2 -6640.681} C_VEL
LIN {X 0,Y 488.694,Z 226.106,A -85,B 0,C 180,E1 -6644.138,E2 -6644.138} C_VEL
LIN {X 0,Y 488.694,Z 226.112,A -85,B 0,C 180,E1 -6646.692,E2 -6646.692} C_VEL
LIN {X 0,Y 488.709,Z 226.111,A -85,B 0,C 180,E1 -6649.22,E2 -6649.22} C_VEL
LIN {X 0,Y 488.833,Z 226.093,A -85,B 0,C 180,E1 -6652.739,E2 -6652.739} C_VEL
LIN {X 0,Y 488.782,Z 226.1,A -85,B 0,C 180,E1 -6655.046,E2 -6655.046} C_VEL
LIN {X 0,Y 488.93,Z 226.082,A -85,B 0,C 180,E1 -6657.523,E2 -6657.523} C_VEL
LIN {X 0,Y 488.946,Z 226.075,A -85,B 0,C 180,E1 -6659.995,E2 -6659.995} C_VEL
LIN {X 0,Y 488.937,Z 226.076,A -85,B 0,C 180,E1 -6662.466,E2 -6662.466} C_VEL
LIN {X 0,Y 488.819,Z 226.096,A -85,B 0,C 180,E1 -6665.77,E2 -6665.77} C_VEL
LIN {X 0,Y 488.793,Z 226.095,A -85,B 0,C 180,E1 -6668.261,E2 -6668.261} C_VEL
LIN {X 0,Y 488.805,Z 226.1,A -85,B 0,C 180,E1 -6671.606,E2 -6671.606} C_VEL
LIN {X 0,Y 488.735,Z 226.104,A -85,B 0,C 180,E1 -6674.995,E2 -6674.995} C_VEL
LIN {X 0,Y 488.721,Z 226.106,A -85,B 0,C 180,E1 -6678.436,E2 -6678.436} C_VEL
LIN {X 0,Y 488.706,Z 226.108,A -85,B 0,C 180,E1 -6681.063,E2 -6681.063} C_VEL
LIN {X 0,Y 488.761,Z 226.154,A -85,B 0,C 180,E1 -6684.185,E2 -6684.185} C_VEL
LIN {X 0,Y 489.173,Z 228.131,A -85,B 0,C 180,E1 -6684.615,E2 -6684.615} C_VEL
LIN {X 0,Y 489.774,Z 232.933,A -85,B 0,C 180,E1 -6685.49,E2 -6685.49} C_VEL
LIN {X 0,Y 489.361,Z 250.4,A -85,B 0,C 180,E1 -6688.555,E2 -6688.555} C_VEL
LIN {X 0,Y 489.301,Z 257.397,A -85,B 0,C 180,E1 -6689.756,E2 -6689.756} C_VEL
LIN {X 0,Y 491.76,Z 272.036,A -85,B 0,C 180,E1 -6690.091,E2 -6690.091} C_VEL
LIN {X 0,Y 491.05,Z 365.914,A -85,B 0,C 180,E1 -6691.529,E2 -6691.529} C_VEL
LIN {X 0,Y 490.785,Z 379.313,A -85,B 0,C 180,E1 -6691.91,E2 -6691.91} C_VEL
LIN {X 0,Y 490.514,Z 390.732,A -85,B 0,C 180,E1 -6692.385,E2 -6692.385} C_VEL
LIN {X 0,Y 490.151,Z 402.04,A -85,B 0,C 180,E1 -6693.006,E2 -6693.006} C_VEL
LIN {X 0,Y 489.718,Z 413.471,A -85,B 0,C 180,E1 -6693.818,E2 -6693.818} C_VEL
LIN {X 0,Y 489.302,Z 424.398,A -85,B 0,C 180,E1 -6694.792,E2 -6694.792} C_VEL
LIN {X 0,Y 488.917,Z 433.919,A -85,B 0,C 180,E1 -6695.848,E2 -6695.848} C_VEL
LIN {X 0,Y 488.582,Z 441.991,A -85,B 0,C 180,E1 -6696.947,E2 -6696.947} C_VEL
LIN {X 0,Y 488.349,Z 449.578,A -85,B 0,C 180,E1 -6698.22,E2 -6698.22} C_VEL
LIN {X 0,Y 488.119,Z 455.827,A -85,B 0,C 180,E1 -6699.535,E2 -6699.535} C_VEL
LIN {X 0,Y 487.99,Z 460.934,A -85,B 0,C 180,E1 -6700.931,E2 -6700.931} C_VEL
LIN {X 0,Y 487.9,Z 464.023,A -85,B 0,C 180,E1 -6702.041,E2 -6702.041} C_VEL
LIN {X 0,Y 487.87,Z 465.518,A -85,B 0,C 180,E1 -6702.723,E2 -6702.723} C_VEL
LIN {X 0,Y 487.812,Z 467.71,A -85,B 0,C 180,E1 -6704.219,E2 -6704.219} C_VEL
LIN {X 0,Y 487.132,Z 468.378,A -85,B 0,C 180,E1 -6704.906,E2 -6704.906} C_VEL
LIN {X 0,Y 484.243,Z 468.802,A -85,B 0,C 180,E1 -6706.025,E2 -6706.025} C_VEL
LIN {X 0,Y 481.82,Z 468.614,A -85,B 0,C 180,E1 -6706.926,E2 -6706.926} C_VEL
LIN {X 0,Y 480.797,Z 468.117,A -85,B 0,C 180,E1 -6707.621,E2 -6707.621} C_VEL
LIN {X 0,Y 480.723,Z 467.874,A -85,B 0,C 180,E1 -6707.855,E2 -6707.855} C_VEL
LIN {X 0,Y 480.774,Z 465.477,A -85,B 0,C 180,E1 -6709.463,E2 -6709.463} C_VEL
LIN {X 0,Y 480.878,Z 461.47,A -85,B 0,C 180,E1 -6711.067,E2 -6711.067} C_VEL
LIN {X 0,Y 481.028,Z 456.793,A -85,B 0,C 180,E1 -6712.414,E2 -6712.414} C_VEL
LIN {X 0,Y 481.25,Z 450.28,A -85,B 0,C 180,E1 -6713.851,E2 -6713.851} C_VEL
LIN {X 0,Y 481.516,Z 443.338,A -85,B 0,C 180,E1 -6715.062,E2 -6715.062} C_VEL
LIN {X 0,Y 481.874,Z 434.222,A -85,B 0,C 180,E1 -6716.345,E2 -6716.345} C_VEL
LIN {X 0,Y 482.238,Z 425.225,A -85,B 0,C 180,E1 -6717.371,E2 -6717.371} C_VEL
LIN {X 0,Y 482.719,Z 414.051,A -85,B 0,C 180,E1 -6718.392,E2 -6718.392} C_VEL
LIN {X 0,Y 483.13,Z 403.135,A -85,B 0,C 180,E1 -6719.19,E2 -6719.19} C_VEL
LIN {X 0,Y 483.544,Z 391.675,A -85,B 0,C 180,E1 -6719.847,E2 -6719.847} C_VEL
LIN {X 0,Y 483.871,Z 378.701,A -85,B 0,C 180,E1 -6720.394,E2 -6720.394} C_VEL
LIN {X 0,Y 484.191,Z 365.738,A -85,B 0,C 180,E1 -6720.761,E2 -6720.761} C_VEL
LIN {X 0,Y 484.799,Z 271.779,A -85,B 0,C 180,E1 -6722.219,E2 -6722.219} C_VEL
LIN {X 0,Y 482.404,Z 258.123,A -85,B 0,C 180,E1 -6722.535,E2 -6722.535} C_VEL
LIN {X 0,Y 482.464,Z 254.664,A -85,B 0,C 180,E1 -6723.157,E2 -6723.157} C_VEL
LIN {X 0,Y 483.07,Z 239.21,A -85,B 0,C 180,E1 -6726.232,E2 -6726.232} C_VEL
LIN {X 0,Y 482.989,Z 233.873,A -85,B 0,C 180,E1 -6727.321,E2 -6727.321} C_VEL
LIN {X 0,Y 481.656,Z 227.048,A -85,B 0,C 180,E1 -6728.834,E2 -6728.834} C_VEL
LIN {X 0,Y 481.631,Z 226.992,A -85,B 0,C 180,E1 -6732.157,E2 -6732.157} C_VEL
LIN {X 0,Y 481.687,Z 226.985,A -85,B 0,C 180,E1 -6734.776,E2 -6734.776} C_VEL
LIN {X 0,Y 481.72,Z 226.978,A -85,B 0,C 180,E1 -6738.216,E2 -6738.216} C_VEL
LIN {X 0,Y 481.693,Z 226.978,A -85,B 0,C 180,E1 -6741.612,E2 -6741.612} C_VEL
LIN {X 0,Y 481.756,Z 226.971,A -85,B 0,C 180,E1 -6744.14,E2 -6744.14} C_VEL
LIN {X 0,Y 481.859,Z 226.959,A -85,B 0,C 180,E1 -6747.494,E2 -6747.494} C_VEL
LIN {X 0,Y 481.859,Z 226.957,A -85,B 0,C 180,E1 -6750.001,E2 -6750.001} C_VEL
LIN {X 0,Y 481.859,Z 226.958,A -85,B 0,C 180,E1 -6752.509,E2 -6752.509} C_VEL
LIN {X 0,Y 481.757,Z 226.971,A -85,B 0,C 180,E1 -6755.862,E2 -6755.862} C_VEL
LIN {X 0,Y 481.696,Z 226.977,A -85,B 0,C 180,E1 -6758.391,E2 -6758.391} C_VEL
LIN {X 0,Y 481.725,Z 226.977,A -85,B 0,C 180,E1 -6761.787,E2 -6761.787} C_VEL
LIN {X 0,Y 481.678,Z 226.984,A -85,B 0,C 180,E1 -6765.228,E2 -6765.228} C_VEL
LIN {X 0,Y 481.642,Z 226.984,A -85,B 0,C 180,E1 -6768.726,E2 -6768.726} C_VEL
LIN {X 0,Y 481.58,Z 226.996,A -85,B 0,C 180,E1 -6771.399,E2 -6771.399} C_VEL
LIN {X 0,Y 481.616,Z 226.992,A -85,B 0,C 180,E1 -6774.118,E2 -6774.118} C_VEL
LIN {X 0,Y 481.689,Z 226.978,A -85,B 0,C 180,E1 -6777.145,E2 -6777.145} C_VEL
LIN {X 0,Y 481.63,Z 226.991,A -85,B 0,C 180,E1 -6779.746,E2 -6779.746} C_VEL
LIN {X 0,Y 481.617,Z 226.989,A -85,B 0,C 180,E1 -6782.68,E2 -6782.68} C_VEL
LIN {X 0,Y 481.588,Z 226.993,A -85,B 0,C 180,E1 -6785.715,E2 -6785.715} C_VEL
LIN {X 0,Y 481.663,Z 226.981,A -85,B 0,C 180,E1 -6789.36,E2 -6789.36} C_VEL
LIN {X 0,Y 481.627,Z 226.991,A -85,B 0,C 180,E1 -6792.164,E2 -6792.164} C_VEL
LIN {X 0,Y 481.615,Z 226.996,A -85,B 0,C 180,E1 -6794.464,E2 -6794.464} C_VEL
LIN {X 0,Y 481.647,Z 226.989,A -85,B 0,C 180,E1 -6796.852,E2 -6796.852} C_VEL
LIN {X 0,Y 481.654,Z 226.984,A -85,B 0,C 180,E1 -6800.068,E2 -6800.068} C_VEL
LIN {X 0,Y 481.594,Z 226.993,A -85,B 0,C 180,E1 -6803.26,E2 -6803.26} C_VEL
LIN {X 0,Y 481.663,Z 226.983,A -85,B 0,C 180,E1 -6806.336,E2 -6806.336} C_VEL
LIN {X 0,Y 481.623,Z 226.99,A -85,B 0,C 180,E1 -6809.424,E2 -6809.424} C_VEL
LIN {X 0,Y 481.675,Z 226.98,A -85,B 0,C 180,E1 -6812.175,E2 -6812.175} C_VEL
LIN {X 0,Y 481.691,Z 226.983,A -85,B 0,C 180,E1 -6814.976,E2 -6814.976} C_VEL
LIN {X 0,Y 481.632,Z 226.988,A -85,B 0,C 180,E1 -6817.711,E2 -6817.711} C_VEL
LIN {X 0,Y 481.69,Z 226.978,A -85,B 0,C 180,E1 -6820.4,E2 -6820.4} C_VEL
LIN {X 0,Y 481.667,Z 226.984,A -85,B 0,C 180,E1 -6823.04,E2 -6823.04} C_VEL
LIN {X 0,Y 481.679,Z 226.988,A -85,B 0,C 180,E1 -6825.645,E2 -6825.645} C_VEL
LIN {X 0,Y 481.745,Z 226.973,A -85,B 0,C 180,E1 -6828.221,E2 -6828.221} C_VEL
LIN {X 0,Y 481.738,Z 226.979,A -85,B 0,C 180,E1 -6831.617,E2 -6831.617} C_VEL
LIN {X 0,Y 481.785,Z 226.971,A -85,B 0,C 180,E1 -6834.145,E2 -6834.145} C_VEL
LIN {X 0,Y 481.92,Z 226.952,A -85,B 0,C 180,E1 -6837.498,E2 -6837.498} C_VEL
LIN {X 0,Y 481.915,Z 226.959,A -85,B 0,C 180,E1 -6840.005,E2 -6840.005} C_VEL
LIN {X 0,Y 481.914,Z 226.954,A -85,B 0,C 180,E1 -6842.513,E2 -6842.513} C_VEL
LIN {X 0,Y 481.787,Z 226.969,A -85,B 0,C 180,E1 -6845.866,E2 -6845.866} C_VEL
LIN {X 0,Y 481.728,Z 226.982,A -85,B 0,C 180,E1 -6848.394,E2 -6848.394} C_VEL
LIN {X 0,Y 481.763,Z 226.97,A -85,B 0,C 180,E1 -6851.789,E2 -6851.789} C_VEL
LIN {X 0,Y 481.753,Z 226.971,A -85,B 0,C 180,E1 -6855.228,E2 -6855.228} C_VEL
LIN {X 0,Y 481.722,Z 226.983,A -85,B 0,C 180,E1 -6858.726,E2 -6858.726} C_VEL
LIN {X 0,Y 481.661,Z 226.983,A -85,B 0,C 180,E1 -6861.398,E2 -6861.398} C_VEL
LIN {X 0,Y 481.664,Z 226.982,A -85,B 0,C 180,E1 -6864.118,E2 -6864.118} C_VEL
LIN {X 0,Y 481.671,Z 226.988,A -85,B 0,C 180,E1 -6867.12,E2 -6867.12} C_VEL
LIN {X 0,Y 481.684,Z 226.98,A -85,B 0,C 180,E1 -6869.745,E2 -6869.745} C_VEL
LIN {X 0,Y 481.67,Z 226.983,A -85,B 0,C 180,E1 -6872.678,E2 -6872.678} C_VEL
LIN {X 0,Y 481.647,Z 226.986,A -85,B 0,C 180,E1 -6875.713,E2 -6875.713} C_VEL
LIN {X 0,Y 481.685,Z 226.981,A -85,B 0,C 180,E1 -6878.862,E2 -6878.862} C_VEL
LIN {X 0,Y 481.634,Z 226.986,A -85,B 0,C 180,E1 -6882.166,E2 -6882.166} C_VEL
LIN {X 0,Y 481.669,Z 226.989,A -85,B 0,C 180,E1 -6885.543,E2 -6885.543} C_VEL
LIN {X 0,Y 481.642,Z 226.984,A -85,B 0,C 180,E1 -6888.956,E2 -6888.956} C_VEL
LIN {X 0,Y 481.653,Z 226.989,A -85,B 0,C 180,E1 -6891.997,E2 -6891.997} C_VEL
LIN {X 0,Y 481.699,Z 226.978,A -85,B 0,C 180,E1 -6895.318,E2 -6895.318} C_VEL
LIN {X 0,Y 481.66,Z 226.989,A -85,B 0,C 180,E1 -6898.311,E2 -6898.311} C_VEL
LIN {X 0,Y 481.691,Z 226.981,A -85,B 0,C 180,E1 -6901.217,E2 -6901.217} C_VEL
LIN {X 0,Y 481.677,Z 226.988,A -85,B 0,C 180,E1 -6904.04,E2 -6904.04} C_VEL
LIN {X 0,Y 481.713,Z 227.178,A -85,B 0,C 180,E1 -6905.486,E2 -6905.486} C_VEL
LIN {X 0,Y 483.451,Z 236.472,A -85,B 0,C 180,E1 -6907.34,E2 -6907.34} C_VEL
LIN {X 0,Y 483.292,Z 244.908,A -85,B 0,C 180,E1 -6908.904,E2 -6908.904} C_VEL
LIN {X 0,Y 482.575,Z 262.977,A -85,B 0,C 180,E1 -6912.19,E2 -6912.19} C_VEL
LIN {X 0,Y 482.343,Z 270.239,A -85,B 0,C 180,E1 -6913.472,E2 -6913.472} C_VEL
LIN {X 0,Y 482.974,Z 274.455,A -85,B 0,C 180,E1 -6913.604,E2 -6913.604} C_VEL
LIN {X 0,Y 484.859,Z 287.137,A -85,B 0,C 180,E1 -6913.864,E2 -6913.864} C_VEL
LIN {X 0,Y 484.167,Z 378.893,A -85,B 0,C 180,E1 -6915.283,E2 -6915.283} C_VEL
LIN {X 0,Y 483.833,Z 392.581,A -85,B 0,C 180,E1 -6915.676,E2 -6915.676} C_VEL
LIN {X 0,Y 483.428,Z 405.425,A -85,B 0,C 180,E1 -6916.227,E2 -6916.227} C_VEL
LIN {X 0,Y 482.975,Z 417.967,A -85,B 0,C 180,E1 -6916.964,E2 -6916.964} C_VEL
LIN {X 0,Y 482.612,Z 429.234,A -85,B 0,C 180,E1 -6917.816,E2 -6917.816} C_VEL
LIN {X 0,Y 482.209,Z 438.207,A -85,B 0,C 180,E1 -6918.651,E2 -6918.651} C_VEL
LIN {X 0,Y 481.803,Z 447.494,A -85,B 0,C 180,E1 -6919.705,E2 -6919.705} C_VEL
LIN {X 0,Y 481.419,Z 456.509,A -85,B 0,C 180,E1 -6920.97,E2 -6920.97} C_VEL
LIN {X 0,Y 481.194,Z 463.769,A -85,B 0,C 180,E1 -6922.234,E2 -6922.234} C_VEL
LIN {X 0,Y 480.994,Z 469.641,A -85,B 0,C 180,E1 -6923.516,E2 -6923.516} C_VEL
LIN {X 0,Y 480.906,Z 474.748,A -85,B 0,C 180,E1 -6924.968,E2 -6924.968} C_VEL
LIN {X 0,Y 480.831,Z 477.056,A -85,B 0,C 180,E1 -6925.808,E2 -6925.808} C_VEL
LIN {X 0,Y 480.875,Z 478.933,A -85,B 0,C 180,E1 -6926.647,E2 -6926.647} C_VEL
LIN {X 0,Y 480.808,Z 480.339,A -85,B 0,C 180,E1 -6927.485,E2 -6927.485} C_VEL
LIN {X 0,Y 480.793,Z 481.34,A -85,B 0,C 180,E1 -6928.323,E2 -6928.323} C_VEL
LIN {X 0,Y 480.763,Z 481.951,A -85,B 0,C 180,E1 -6929.161,E2 -6929.161} C_VEL
LIN {X 0,Y 480.746,Z 482.169,A -85,B 0,C 180,E1 -6929.999,E2 -6929.999} C_VEL
LIN {X 0,Y 480.763,Z 481.952,A -85,B 0,C 180,E1 -6930.836,E2 -6930.836} C_VEL
LIN {X 0,Y 480.793,Z 481.341,A -85,B 0,C 180,E1 -6931.674,E2 -6931.674} C_VEL
LIN {X 0,Y 480.807,Z 480.339,A -85,B 0,C 180,E1 -6932.512,E2 -6932.512} C_VEL
LIN {X 0,Y 480.874,Z 478.934,A -85,B 0,C 180,E1 -6933.35,E2 -6933.35} C_VEL
LIN {X 0,Y 480.842,Z 475.98,A -85,B 0,C 180,E1 -6934.609,E2 -6934.609} C_VEL
LIN {X 0,Y 480.961,Z 471.982,A -85,B 0,C 180,E1 -6935.869,E2 -6935.869} C_VEL
LIN {X 0,Y 481.114,Z 465.827,A -85,B 0,C 180,E1 -6937.342,E2 -6937.342} C_VEL
LIN {X 0,Y 481.341,Z 459.103,A -85,B 0,C 180,E1 -6938.606,E2 -6938.606} C_VEL
LIN {X 0,Y 481.683,Z 450.758,A -85,B 0,C 180,E1 -6939.87,E2 -6939.87} C_VEL
LIN {X 0,Y 482.008,Z 442.174,A -85,B 0,C 180,E1 -6940.925,E2 -6940.925} C_VEL
LIN {X 0,Y 482.488,Z 431.579,A -85,B 0,C 180,E1 -6941.978,E2 -6941.978} C_VEL
LIN {X 0,Y 482.879,Z 420.147,A -85,B 0,C 180,E1 -6942.892,E2 -6942.892} C_VEL
LIN {X 0,Y 483.287,Z 409.512,A -85,B 0,C 180,E1 -6943.56,E2 -6943.56} C_VEL
LIN {X 0,Y 483.668,Z 397.525,A -85,B 0,C 180,E1 -6944.139,E2 -6944.139} C_VEL
LIN {X 0,Y 484.038,Z 384.597,A -85,B 0,C 180,E1 -6944.584,E2 -6944.584} C_VEL
LIN {X 0,Y 484.264,Z 370.906,A -85,B 0,C 180,E1 -6944.872,E2 -6944.872} C_VEL
LIN {X 0,Y 484.831,Z 285.495,A -85,B 0,C 180,E1 -6946.184,E2 -6946.184} C_VEL
LIN {X 0,Y 482.285,Z 270.101,A -85,B 0,C 180,E1 -6946.538,E2 -6946.538} C_VEL
LIN {X 0,Y 482.794,Z 255.186,A -85,B 0,C 180,E1 -6949.134,E2 -6949.134} C_VEL
LIN {X 0,Y 483.397,Z 238.005,A -85,B 0,C 180,E1 -6952.208,E2 -6952.208} C_VEL
LIN {X 0,Y 482.864,Z 233.047,A -85,B 0,C 180,E1 -6953.138,E2 -6953.138} C_VEL
LIN {X 0,Y 481.692,Z 227.104,A -85,B 0,C 180,E1 -6954.34,E2 -6954.34} C_VEL
LIN {X 0,Y 481.722,Z 226.98,A -85,B 0,C 180,E1 -6957.129,E2 -6957.129} C_VEL
LIN {X 0,Y 481.683,Z 226.988,A -85,B 0,C 180,E1 -6959.739,E2 -6959.739} C_VEL
LIN {X 0,Y 481.677,Z 226.983,A -85,B 0,C 180,E1 -6962.672,E2 -6962.672} C_VEL
LIN {X 0,Y 481.636,Z 226.992,A -85,B 0,C 180,E1 -6965.707,E2 -6965.707} C_VEL
LIN {X 0,Y 481.669,Z 226.982,A -85,B 0,C 180,E1 -6968.857,E2 -6968.857} C_VEL
LIN {X 0,Y 481.628,Z 226.995,A -85,B 0,C 180,E1 -6972.16,E2 -6972.16} C_VEL
LIN {X 0,Y 481.656,Z 226.984,A -85,B 0,C 180,E1 -6975.538,E2 -6975.538} C_VEL
LIN {X 0,Y 481.625,Z 226.989,A -85,B 0,C 180,E1 -6978.951,E2 -6978.951} C_VEL
LIN {X 0,Y 481.63,Z 226.99,A -85,B 0,C 180,E1 -6981.993,E2 -6981.993} C_VEL
LIN {X 0,Y 481.678,Z 226.981,A -85,B 0,C 180,E1 -6985.313,E2 -6985.313} C_VEL
LIN {X 0,Y 481.638,Z 226.991,A -85,B 0,C 180,E1 -6988.307,E2 -6988.307} C_VEL
LIN {X 0,Y 481.654,Z 226.985,A -85,B 0,C 180,E1 -6991.212,E2 -6991.212} C_VEL
LIN {X 0,Y 481.624,Z 226.985,A -85,B 0,C 180,E1 -6994.034,E2 -6994.034} C_VEL
LIN {X 0,Y 481.647,Z 226.988,A -85,B 0,C 180,E1 -6996.814,E2 -6996.814} C_VEL
LIN {X 0,Y 481.659,Z 226.983,A -85,B 0,C 180,E1 -6999.497,E2 -6999.497} C_VEL
LIN {X 0,Y 481.644,Z 226.985,A -85,B 0,C 180,E1 -7002.152,E2 -7002.152} C_VEL
LIN {X 0,Y 481.712,Z 226.98,A -85,B 0,C 180,E1 -7004.77,E2 -7004.77} C_VEL
LIN {X 0,Y 481.737,Z 226.971,A -85,B 0,C 180,E1 -7008.21,E2 -7008.21} C_VEL
LIN {X 0,Y 481.707,Z 226.979,A -85,B 0,C 180,E1 -7011.606,E2 -7011.606} C_VEL
LIN {X 0,Y 481.78,Z 226.966,A -85,B 0,C 180,E1 -7014.134,E2 -7014.134} C_VEL
LIN {X 0,Y 481.897,Z 226.958,A -85,B 0,C 180,E1 -7017.487,E2 -7017.487} C_VEL
LIN {X 0,Y 481.917,Z 226.95,A -85,B 0,C 180,E1 -7019.995,E2 -7019.995} C_VEL
LIN {X 0,Y 481.904,Z 226.952,A -85,B 0,C 180,E1 -7022.502,E2 -7022.502} C_VEL
LIN {X 0,Y 481.778,Z 226.972,A -85,B 0,C 180,E1 -7025.855,E2 -7025.855} C_VEL
LIN {X 0,Y 481.738,Z 226.974,A -85,B 0,C 180,E1 -7028.383,E2 -7028.383} C_VEL
LIN {X 0,Y 481.768,Z 226.975,A -85,B 0,C 180,E1 -7031.778,E2 -7031.778} C_VEL
LIN {X 0,Y 481.714,Z 226.981,A -85,B 0,C 180,E1 -7035.218,E2 -7035.218} C_VEL
LIN {X 0,Y 481.678,Z 226.983,A -85,B 0,C 180,E1 -7038.716,E2 -7038.716} C_VEL
LIN {X 0,Y 481.642,Z 226.991,A -85,B 0,C 180,E1 -7041.387,E2 -7041.387} C_VEL
LIN {X 0,Y 481.737,Z 227.108,A -85,B 0,C 180,E1 -7044.045,E2 -7044.045} C_VEL
LIN {X 0,Y 482.814,Z 233.268,A -85,B 0,C 180,E1 -7045.238,E2 -7045.238} C_VEL
LIN {X 0,Y 482.411,Z 250.228,A -85,B 0,C 180,E1 -7048.252,E2 -7048.252} C_VEL
LIN {X 0,Y 482.324,Z 257.551,A -85,B 0,C 180,E1 -7049.512,E2 -7049.512} C_VEL
LIN {X 0,Y 484.96,Z 273.037,A -85,B 0,C 180,E1 -7049.87,E2 -7049.87} C_VEL
LIN {X 0,Y 484.167,Z 365.917,A -85,B 0,C 180,E1 -7051.317,E2 -7051.317} C_VEL
LIN {X 0,Y 483.897,Z 379.619,A -85,B 0,C 180,E1 -7051.714,E2 -7051.714} C_VEL
LIN {X 0,Y 483.582,Z 392.532,A -85,B 0,C 180,E1 -7052.274,E2 -7052.274} C_VEL
LIN {X 0,Y 483.195,Z 403.663,A -85,B 0,C 180,E1 -7052.921,E2 -7052.921} C_VEL
LIN {X 0,Y 482.705,Z 414.758,A -85,B 0,C 180,E1 -7053.739,E2 -7053.739} C_VEL
LIN {X 0,Y 482.27,Z 425.575,A -85,B 0,C 180,E1 -7054.739,E2 -7054.739} C_VEL
LIN {X 0,Y 481.864,Z 434.862,A -85,B 0,C 180,E1 -7055.809,E2 -7055.809} C_VEL
LIN {X 0,Y 481.525,Z 443.325,A -85,B 0,C 180,E1 -7057.007,E2 -7057.007} C_VEL
LIN {X 0,Y 481.239,Z 451.164,A -85,B 0,C 180,E1 -7058.393,E2 -7058.393} C_VEL
LIN {X 0,Y 481.032,Z 456.586,A -85,B 0,C 180,E1 -7059.602,E2 -7059.602} C_VEL
LIN {X 0,Y 480.9,Z 461.784,A -85,B 0,C 180,E1 -7061.109,E2 -7061.109} C_VEL
LIN {X 0,Y 480.787,Z 464.703,A -85,B 0,C 180,E1 -7062.243,E2 -7062.243} C_VEL
LIN {X 0,Y 480.712,Z 466.862,A -85,B 0,C 180,E1 -7063.393,E2 -7063.393} C_VEL
LIN {X 0,Y 480.736,Z 468.213,A -85,B 0,C 180,E1 -7064.554,E2 -7064.554} C_VEL
LIN {X 0,Y 480.709,Z 468.802,A -85,B 0,C 180,E1 -7065.745,E2 -7065.745} C_VEL
LIN {X 0,Y 480.673,Z 468.584,A -85,B 0,C 180,E1 -7066.963,E2 -7066.963} C_VEL
LIN {X 0,Y 480.723,Z 467.874,A -85,B 0,C 180,E1 -7067.855,E2 -7067.855} C_VEL
LIN {X 0,Y 480.079,Z 467.053,A -85,B 0,C 180,E1 -7068.547,E2 -7068.547} C_VEL
LIN {X 0,Y 477.238,Z 465.155,A -85,B 0,C 180,E1 -7069.661,E2 -7069.661} C_VEL
LIN {X 0,Y 474.863,Z 463.169,A -85,B 0,C 180,E1 -7070.546,E2 -7070.546} C_VEL
LIN {X 0,Y 473.898,Z 461.322,A -85,B 0,C 180,E1 -7071.219,E2 -7071.219} C_VEL
LIN {X 0,Y 473.85,Z 460.634,A -85,B 0,C 180,E1 -7071.445,E2 -7071.445} C_VEL
LIN {X 0,Y 474.025,Z 455.286,A -85,B 0,C 180,E1 -7072.897,E2 -7072.897} C_VEL
LIN {X 0,Y 474.309,Z 448.156,A -85,B 0,C 180,E1 -7074.384,E2 -7074.384} C_VEL
LIN {X 0,Y 474.564,Z 441.47,A -85,B 0,C 180,E1 -7075.499,E2 -7075.499} C_VEL
LIN {X 0,Y 474.953,Z 432.804,A -85,B 0,C 180,E1 -7076.68,E2 -7076.68} C_VEL
LIN {X 0,Y 475.379,Z 422.179,A -85,B 0,C 180,E1 -7077.846,E2 -7077.846} C_VEL
LIN {X 0,Y 475.827,Z 411.937,A -85,B 0,C 180,E1 -7078.75,E2 -7078.75} C_VEL
LIN {X 0,Y 476.306,Z 399.93,A -85,B 0,C 180,E1 -7079.585,E2 -7079.585} C_VEL
LIN {X 0,Y 476.801,Z 387.05,A -85,B 0,C 180,E1 -7080.266,E2 -7080.266} C_VEL
LIN {X 0,Y 477.087,Z 373.908,A -85,B 0,C 180,E1 -7080.759,E2 -7080.759} C_VEL
LIN {X 0,Y 477.33,Z 360.873,A -85,B 0,C 180,E1 -7081.068,E2 -7081.068} C_VEL
LIN {X 0,Y 477.873,Z 272.154,A -85,B 0,C 180,E1 -7082.45,E2 -7082.45} C_VEL
LIN {X 0,Y 475.5,Z 258.535,A -85,B 0,C 180,E1 -7082.762,E2 -7082.762} C_VEL
LIN {X 0,Y 475.431,Z 257.649,A -85,B 0,C 180,E1 -7082.847,E2 -7082.847} C_VEL
LIN {X 0,Y 476.094,Z 240.839,A -85,B 0,C 180,E1 -7086.216,E2 -7086.216} C_VEL
LIN {X 0,Y 476.147,Z 236.026,A -85,B 0,C 180,E1 -7087.206,E2 -7087.206} C_VEL
LIN {X 0,Y 474.614,Z 227.906,A -85,B 0,C 180,E1 -7089.024,E2 -7089.024} C_VEL
LIN {X 0,Y 474.58,Z 227.87,A -85,B 0,C 180,E1 -7091.883,E2 -7091.883} C_VEL
LIN {X 0,Y 474.64,Z 227.865,A -85,B 0,C 180,E1 -7094.544,E2 -7094.544} C_VEL
LIN {X 0,Y 474.662,Z 227.855,A -85,B 0,C 180,E1 -7098.038,E2 -7098.038} C_VEL
LIN {X 0,Y 474.658,Z 227.854,A -85,B 0,C 180,E1 -7101.487,E2 -7101.487} C_VEL
LIN {X 0,Y 474.715,Z 227.847,A -85,B 0,C 180,E1 -7104.053,E2 -7104.053} C_VEL
LIN {X 0,Y 474.826,Z 227.835,A -85,B 0,C 180,E1 -7107.457,E2 -7107.457} C_VEL
LIN {X 0,Y 474.831,Z 227.832,A -85,B 0,C 180,E1 -7110.001,E2 -7110.001} C_VEL
LIN {X 0,Y 474.826,Z 227.835,A -85,B 0,C 180,E1 -7112.546,E2 -7112.546} C_VEL
LIN {X 0,Y 474.717,Z 227.847,A -85,B 0,C 180,E1 -7115.95,E2 -7115.95} C_VEL
LIN {X 0,Y 474.661,Z 227.854,A -85,B 0,C 180,E1 -7118.516,E2 -7118.516} C_VEL
LIN {X 0,Y 474.667,Z 227.855,A -85,B 0,C 180,E1 -7121.965,E2 -7121.965} C_VEL
LIN {X 0,Y 474.633,Z 227.865,A -85,B 0,C 180,E1 -7125.459,E2 -7125.459} C_VEL
LIN {X 0,Y 474.595,Z 227.863,A -85,B 0,C 180,E1 -7129.014,E2 -7129.014} C_VEL
LIN {X 0,Y 474.525,Z 227.88,A -85,B 0,C 180,E1 -7131.733,E2 -7131.733} C_VEL
LIN {X 0,Y 474.598,Z 227.862,A -85,B 0,C 180,E1 -7134.497,E2 -7134.497} C_VEL
LIN {X 0,Y 474.637,Z 227.858,A -85,B 0,C 180,E1 -7137.344,E2 -7137.344} C_VEL
LIN {X 0,Y 474.554,Z 227.867,A -85,B 0,C 180,E1 -7140.817,E2 -7140.817} C_VEL
LIN {X 0,Y 474.583,Z 227.87,A -85,B 0,C 180,E1 -7143.99,E2 -7143.99} C_VEL
LIN {X 0,Y 474.52,Z 227.872,A -85,B 0,C 180,E1 -7146.906,E2 -7146.906} C_VEL
LIN {X 0,Y 474.6,Z 227.862,A -85,B 0,C 180,E1 -7149.657,E2 -7149.657} C_VEL
LIN {X 0,Y 474.605,Z 227.863,A -85,B 0,C 180,E1 -7152.937,E2 -7152.937} C_VEL
LIN {X 0,Y 474.575,Z 227.865,A -85,B 0,C 180,E1 -7155.903,E2 -7155.903} C_VEL
LIN {X 0,Y 474.608,Z 227.864,A -85,B 0,C 180,E1 -7159.045,E2 -7159.045} C_VEL
LIN {X 0,Y 474.582,Z 227.863,A -85,B 0,C 180,E1 -7161.71,E2 -7161.71} C_VEL
LIN {X 0,Y 474.595,Z 227.869,A -85,B 0,C 180,E1 -7164.733,E2 -7164.733} C_VEL
LIN {X 0,Y 474.605,Z 227.861,A -85,B 0,C 180,E1 -7167.795,E2 -7167.795} C_VEL
LIN {X 0,Y 474.598,Z 227.868,A -85,B 0,C 180,E1 -7170.892,E2 -7170.892} C_VEL
LIN {X 0,Y 474.636,Z 227.859,A -85,B 0,C 180,E1 -7173.635,E2 -7173.635} C_VEL
LIN {X 0,Y 474.618,Z 227.86,A -85,B 0,C 180,E1 -7176.648,E2 -7176.648} C_VEL
LIN {X 0,Y 474.64,Z 227.857,A -85,B 0,C 180,E1 -7180.096,E2 -7180.096} C_VEL
LIN {X 0,Y 474.626,Z 227.859,A -85,B 0,C 180,E1 -7182.781,E2 -7182.781} C_VEL
LIN {X 0,Y 474.638,Z 227.863,A -85,B 0,C 180,E1 -7185.427,E2 -7185.427} C_VEL
LIN {X 0,Y 474.699,Z 227.852,A -85,B 0,C 180,E1 -7188.044,E2 -7188.044} C_VEL
LIN {X 0,Y 474.709,Z 227.852,A -85,B 0,C 180,E1 -7191.492,E2 -7191.492} C_VEL
LIN {X 0,Y 474.748,Z 227.849,A -85,B 0,C 180,E1 -7194.058,E2 -7194.058} C_VEL
LIN {X 0,Y 474.886,Z 227.828,A -85,B 0,C 180,E1 -7197.461,E2 -7197.461} C_VEL
LIN {X 0,Y 474.884,Z 227.834,A -85,B 0,C 180,E1 -7200.006,E2 -7200.006} C_VEL
LIN {X 0,Y 474.879,Z 227.83,A -85,B 0,C 180,E1 -7202.55,E2 -7202.55} C_VEL
LIN {X 0,Y 474.75,Z 227.847,A -85,B 0,C 180,E1 -7205.953,E2 -7205.953} C_VEL
LIN {X 0,Y 474.678,Z 227.858,A -85,B 0,C 180,E1 -7208.519,E2 -7208.519} C_VEL
LIN {X 0,Y 474.717,Z 227.849,A -85,B 0,C 180,E1 -7211.967,E2 -7211.967} C_VEL
LIN {X 0,Y 474.695,Z 227.85,A -85,B 0,C 180,E1 -7215.771,E2 -7215.771} C_VEL
LIN {X 0,Y 474.676,Z 227.856,A -85,B 0,C 180,E1 -7219.014,E2 -7219.014} C_VEL
LIN {X 0,Y 474.604,Z 227.861,A -85,B 0,C 180,E1 -7221.733,E2 -7221.733} C_VEL
LIN {X 0,Y 474.643,Z 227.859,A -85,B 0,C 180,E1 -7224.498,E2 -7224.498} C_VEL
LIN {X 0,Y 474.618,Z 227.863,A -85,B 0,C 180,E1 -7227.329,E2 -7227.329} C_VEL
LIN {X 0,Y 474.613,Z 227.86,A -85,B 0,C 180,E1 -7230.234,E2 -7230.234} C_VEL
LIN {X 0,Y 474.634,Z 227.866,A -85,B 0,C 180,E1 -7233.225,E2 -7233.225} C_VEL
LIN {X 0,Y 474.601,Z 227.861,A -85,B 0,C 180,E1 -7236.326,E2 -7236.326} C_VEL
LIN {X 0,Y 474.642,Z 227.863,A -85,B 0,C 180,E1 -7239.55,E2 -7239.55} C_VEL
LIN {X 0,Y 474.594,Z 227.862,A -85,B 0,C 180,E1 -7242.231,E2 -7242.231} C_VEL
LIN {X 0,Y 474.629,Z 227.862,A -85,B 0,C 180,E1 -7245.3,E2 -7245.3} C_VEL
LIN {X 0,Y 474.61,Z 227.862,A -85,B 0,C 180,E1 -7248.212,E2 -7248.212} C_VEL
LIN {X 0,Y 474.637,Z 227.857,A -85,B 0,C 180,E1 -7250.452,E2 -7250.452} C_VEL
LIN {X 0,Y 474.599,Z 227.867,A -85,B 0,C 180,E1 -7253.676,E2 -7253.676} C_VEL
LIN {X 0,Y 474.633,Z 227.857,A -85,B 0,C 180,E1 -7256.778,E2 -7256.778} C_VEL
LIN {X 0,Y 474.618,Z 227.863,A -85,B 0,C 180,E1 -7259.77,E2 -7259.77} C_VEL
LIN {X 0,Y 474.656,Z 227.861,A -85,B 0,C 180,E1 -7262.676,E2 -7262.676} C_VEL
LIN {X 0,Y 474.678,Z 228.007,A -85,B 0,C 180,E1 -7265.274,E2 -7265.274} C_VEL
LIN {X 0,Y 476.456,Z 237.563,A -85,B 0,C 180,E1 -7267.218,E2 -7267.218} C_VEL
LIN {X 0,Y 476.409,Z 244.792,A -85,B 0,C 180,E1 -7268.584,E2 -7268.584} C_VEL
LIN {X 0,Y 475.625,Z 262.863,A -85,B 0,C 180,E1 -7271.921,E2 -7271.921} C_VEL
LIN {X 0,Y 475.393,Z 270.344,A -85,B 0,C 180,E1 -7273.245,E2 -7273.245} C_VEL
LIN {X 0,Y 477.071,Z 280.644,A -85,B 0,C 180,E1 -7273.498,E2 -7273.498} C_VEL
LIN {X 0,Y 478.031,Z 287.658,A -85,B 0,C 180,E1 -7273.642,E2 -7273.642} C_VEL
LIN {X 0,Y 477.308,Z 378.469,A -85,B 0,C 180,E1 -7275.067,E2 -7275.067} C_VEL
LIN {X 0,Y 476.935,Z 392.257,A -85,B 0,C 180,E1 -7275.464,E2 -7275.464} C_VEL
LIN {X 0,Y 476.496,Z 405.178,A -85,B 0,C 180,E1 -7276.022,E2 -7276.022} C_VEL
LIN {X 0,Y 476.031,Z 417.75,A -85,B 0,C 180,E1 -7276.77,E2 -7276.77} C_VEL
LIN {X 0,Y 475.693,Z 427.566,A -85,B 0,C 180,E1 -7277.512,E2 -7277.512} C_VEL
LIN {X 0,Y 475.217,Z 438.032,A -85,B 0,C 180,E1 -7278.482,E2 -7278.482} C_VEL
LIN {X 0,Y 474.769,Z 447.339,A -85,B 0,C 180,E1 -7279.551,E2 -7279.551} C_VEL
LIN {X 0,Y 474.375,Z 456.366,A -85,B 0,C 180,E1 -7280.834,E2 -7280.834} C_VEL
LIN {X 0,Y 474.116,Z 463.636,A -85,B 0,C 180,E1 -7282.118,E2 -7282.118} C_VEL
LIN {X 0,Y 473.894,Z 469.998,A -85,B 0,C 180,E1 -7283.544,E2 -7283.544} C_VEL
LIN {X 0,Y 473.841,Z 474.635,A -85,B 0,C 180,E1 -7284.893,E2 -7284.893} C_VEL
LIN {X 0,Y 473.738,Z 476.946,A -85,B 0,C 180,E1 -7285.745,E2 -7285.745} C_VEL
LIN {X 0,Y 473.769,Z 478.826,A -85,B 0,C 180,E1 -7286.597,E2 -7286.597} C_VEL
LIN {X 0,Y 473.727,Z 480.236,A -85,B 0,C 180,E1 -7287.448,E2 -7287.448} C_VEL
LIN {X 0,Y 473.692,Z 481.851,A -85,B 0,C 180,E1 -7289.148,E2 -7289.148} C_VEL
LIN {X 0,Y 473.673,Z 482.071,A -85,B 0,C 180,E1 -7289.999,E2 -7289.999} C_VEL
LIN {X 0,Y 473.692,Z 481.855,A -85,B 0,C 180,E1 -7290.849,E2 -7290.849} C_VEL
LIN {X 0,Y 473.726,Z 480.241,A -85,B 0,C 180,E1 -7292.549,E2 -7292.549} C_VEL
LIN {X 0,Y 473.769,Z 478.835,A -85,B 0,C 180,E1 -7293.4,E2 -7293.4} C_VEL
LIN {X 0,Y 473.766,Z 475.879,A -85,B 0,C 180,E1 -7294.678,E2 -7294.678} C_VEL
LIN {X 0,Y 473.865,Z 471.878,A -85,B 0,C 180,E1 -7295.958,E2 -7295.958} C_VEL
LIN {X 0,Y 474.035,Z 465.716,A -85,B 0,C 180,E1 -7297.452,E2 -7297.452} C_VEL
LIN {X 0,Y 474.309,Z 458.986,A -85,B 0,C 180,E1 -7298.734,E2 -7298.734} C_VEL
LIN {X 0,Y 474.662,Z 450.639,A -85,B 0,C 180,E1 -7300.017,E2 -7300.017} C_VEL
LIN {X 0,Y 475.021,Z 442.059,A -85,B 0,C 180,E1 -7301.088,E2 -7301.088} C_VEL
LIN {X 0,Y 475.516,Z 431.677,A -85,B 0,C 180,E1 -7302.138,E2 -7302.138} C_VEL
LIN {X 0,Y 475.9,Z 421.271,A -85,B 0,C 180,E1 -7302.992,E2 -7302.992} C_VEL
LIN {X 0,Y 476.368,Z 409.433,A -85,B 0,C 180,E1 -7303.761,E2 -7303.761} C_VEL
LIN {X 0,Y 476.791,Z 397.462,A -85,B 0,C 180,E1 -7304.347,E2 -7304.347} C_VEL
LIN {X 0,Y 477.18,Z 384.557,A -85,B 0,C 180,E1 -7304.798,E2 -7304.798} C_VEL
LIN {X 0,Y 477.415,Z 370.951,A -85,B 0,C 180,E1 -7305.091,E2 -7305.091} C_VEL
LIN {X 0,Y 478.062,Z 286.438,A -85,B 0,C 180,E1 -7306.409,E2 -7306.409} C_VEL
LIN {X 0,Y 475.331,Z 269.992,A -85,B 0,C 180,E1 -7306.795,E2 -7306.795} C_VEL
LIN {X 0,Y 475.831,Z 255.466,A -85,B 0,C 180,E1 -7309.363,E2 -7309.363} C_VEL
LIN {X 0,Y 476.462,Z 239.167,A -85,B 0,C 180,E1 -7312.321,E2 -7312.321} C_VEL
LIN {X 0,Y 475.65,Z 232.968,A -85,B 0,C 180,E1 -7313.51,E2 -7313.51} C_VEL
LIN {X 0,Y 474.651,Z 227.962,A -85,B 0,C 180,E1 -7314.55,E2 -7314.55} C_VEL
LIN {X 0,Y 474.682,Z 227.859,A -85,B 0,C 180,E1 -7317.33,E2 -7317.33} C_VEL
